(*Table Error*)
IF dwMask = 16#4A THEN
	stGroupMessage := 'Table Error: ';
	IF NC_Error_Code = 16#4A00 THEN
		stErrorMessage := 'Table ID not allowed';
	END_IF
	IF NC_Error_Code = 16#4A01 THEN
		stErrorMessage := 'Table type not allowed';
	END_IF
	IF NC_Error_Code = 16#4A02 THEN
		stErrorMessage := 'Number of lines in the table not allowed';
	END_IF
	IF NC_Error_Code = 16#4A03 THEN
		stErrorMessage := 'Number of columns in the table is not allowed';
	END_IF
	IF NC_Error_Code = 16#4A04 THEN
		stErrorMessage := 'Step size (position delta) not allowed';
	END_IF
	IF NC_Error_Code = 16#4A05 THEN
		stErrorMessage := 'Period not allowed';
	END_IF
	IF NC_Error_Code = 16#4A06 THEN
		stErrorMessage := 'Table is not monotonic';
	END_IF
	IF NC_Error_Code = 16#4A07 THEN
		stErrorMessage := 'Table sub type is not allowed';
	END_IF
	IF NC_Error_Code = 16#4A08 THEN
		stErrorMessage := 'Table interpolation type is not allowed';
	END_IF
	IF NC_Error_Code = 16#4A09 THEN
		stErrorMessage := 'Incorrect table main type';
	END_IF
	IF NC_Error_Code = 16#4A10 THEN
		stErrorMessage := 'Table initialisation';
	END_IF
	IF NC_Error_Code = 16#4A11 THEN
		stErrorMessage := 'Not enough memory';
	END_IF
	IF NC_Error_Code = 16#4A12 THEN
		stErrorMessage := 'Function not executed, function not available';
	END_IF
	IF NC_Error_Code = 16#4A13 THEN
		stErrorMessage := 'Line index not allowed';
	END_IF
	IF NC_Error_Code = 16#4A14 THEN
		stErrorMessage := 'Column index not allowed';
	END_IF
	IF NC_Error_Code = 16#4A15 THEN
		stErrorMessage := 'Number of lines not allowed';
	END_IF
	IF NC_Error_Code = 16#4A16 THEN
		stErrorMessage := 'Number of columns not allowed';
	END_IF
	IF NC_Error_Code = 16#4A17 THEN
		stErrorMessage := 'Error in scaling or in range entry';
	END_IF
	IF NC_Error_Code = 16#4A18 THEN
		stErrorMessage := 'Multi table slave out of range';
	END_IF
	IF NC_Error_Code = 16#4A19 THEN
		stErrorMessage := 'Solo table underflow';
	END_IF
	IF NC_Error_Code = 16#4A1B THEN
		stErrorMessage := 'Incorrect execution mode';
	END_IF
	IF NC_Error_Code = 16#4A1C THEN
		stErrorMessage := 'Impermissible parameter';
	END_IF
	IF NC_Error_Code = 16#4A1D THEN
		stErrorMessage := 'Fifo is empty';
	END_IF
	IF NC_Error_Code = 16#4A1E THEN
		stErrorMessage := 'Fifo is full';
	END_IF
	IF NC_Error_Code = 16#4A1F THEN
		stErrorMessage := 'Point-Index of Motion Function invalid';
	END_IF
	IF NC_Error_Code = 16#4A20 THEN
		stErrorMessage := 'No diagonalisation of  matrix';
	END_IF
	IF NC_Error_Code = 16#4A21 THEN
		stErrorMessage := 'Number of spline points to less';
	END_IF
	IF NC_Error_Code = 16#4A22 THEN
		stErrorMessage := 'Fifo must not be overwritten';
	END_IF
END_IF

(*NC-PLC Error*)
IF dwMask = 16#4B THEN
	stGroupMessage := 'NC-PLC Error: ';
	IF NC_Error_Code = 16#4B00 THEN
		stErrorMessage := 'Axis has been stopped';
	END_IF
	IF NC_Error_Code = 16#4B01 THEN
		stErrorMessage := 'Axis cannot be started';
	END_IF
	IF NC_Error_Code = 16#4B02 THEN
		stErrorMessage := 'Control mode not allowed';
	END_IF
	IF NC_Error_Code = 16#4B03 THEN
		stErrorMessage := 'Axis is not moving';
	END_IF
	IF NC_Error_Code = 16#4B04 THEN
		stErrorMessage := 'Wrong mode for RestartPosAndVelo';
	END_IF
	IF NC_Error_Code = 16#4B05 THEN
		stErrorMessage := 'Command not allowed';
	END_IF
	IF NC_Error_Code = 16#4B06 THEN
		stErrorMessage := 'Parameter not correct';
	END_IF
	IF NC_Error_Code = 16#4B07 THEN
		stErrorMessage := 'Timeout axis function block';
	END_IF
	IF NC_Error_Code = 16#4B08 THEN
		stErrorMessage := 'Axis in protected mode';
	END_IF
	IF NC_Error_Code = 16#4B09 THEN
		stErrorMessage := 'Axis is not ready';
	END_IF
	IF NC_Error_Code = 16#4B0A THEN
		stErrorMessage := 'Homing error';
	END_IF
	IF NC_Error_Code = 16#4B0B THEN
		stErrorMessage := 'Invalid definition trigger input definition';
	END_IF
	IF NC_Error_Code = 16#4B0C THEN
		stErrorMessage := 'position latch has been deactivated';
	END_IF
	IF NC_Error_Code = 16#4B0E THEN
		stErrorMessage := 'Supplement not installed';
	END_IF
	IF NC_Error_Code = 16#4B0F THEN
		stErrorMessage := 'Timeout Register Access';
	END_IF
	IF NC_Error_Code = 16#4B10 THEN
		stErrorMessage := 'M-Function request missing';
	END_IF
	IF NC_Error_Code = 16#4B11 THEN
		stErrorMessage := 'Zero shift index is out of range';
	END_IF
	IF NC_Error_Code = 16#4B12 THEN
		stErrorMessage := 'R parameter index or size is invalid';
	END_IF
	IF NC_Error_Code = 16#4B13 THEN
		stErrorMessage := 'Index for tool description is invalid';
	END_IF
	IF NC_Error_Code = 16#4B14 THEN
		stErrorMessage := 'Version of cyclic channel interface does not match to the requested function and function block, resp.';
	END_IF
	IF NC_Error_Code = 16#4B15 THEN
		stErrorMessage := 'Channel is not ready for requested function';
	END_IF
	IF NC_Error_Code = 16#4B16 THEN
		stErrorMessage := 'Requested function is not turned on';
	END_IF
	IF NC_Error_Code = 16#4B20 THEN
		stErrorMessage := 'Cannot append all axes';
	END_IF
	IF NC_Error_Code = 16#4B30 THEN
		stErrorMessage := 'Pointer invalid';
	END_IF
	IF NC_Error_Code = 16#4B31 THEN
		stErrorMessage := 'Size of  memory invalid';
	END_IF
	IF NC_Error_Code = 16#4B32 THEN
		stErrorMessage := 'Invalid cam table ID';
	END_IF
	IF NC_Error_Code = 16#4B33 THEN
		stErrorMessage := 'Invalid point ID';
	END_IF
	IF NC_Error_Code = 16#4B34 THEN
		stErrorMessage := 'Invalid number of points ';
	END_IF
	IF NC_Error_Code = 16#4B35 THEN
		stErrorMessage := 'Invalid MC table type';
	END_IF
	IF NC_Error_Code = 16#4B36 THEN
		stErrorMessage := 'Invalid number of rows';
	END_IF
	IF NC_Error_Code = 16#4B37 THEN
		stErrorMessage := 'Invalid number of columns';
	END_IF
	IF NC_Error_Code = 16#4B38 THEN
		stErrorMessage := 'Invalid Increment';
	END_IF
	IF NC_Error_Code = 16#4B40 THEN
		stErrorMessage := 'Unsupported Terminal Type';
	END_IF
	IF NC_Error_Code = 16#4B41 THEN
		stErrorMessage := 'Register Read/Write Error';
	END_IF
	IF NC_Error_Code = 16#4B42 THEN
		stErrorMessage := 'Axis is Enabled';
	END_IF
	IF NC_Error_Code = 16#4B60 THEN
		stErrorMessage := 'Motion command not be activated';
	END_IF
	IF NC_Error_Code = 16#4B61 THEN
		stErrorMessage := 'Motion command could not be monitored by the PLC';
	END_IF
	IF NC_Error_Code = 16#4B62 THEN
		stErrorMessage := 'Buffered command finished with error';
	END_IF
	IF NC_Error_Code = 16#4B63 THEN
		stErrorMessage := 'Buffered command finished without state feedback';
	END_IF
	IF NC_Error_Code = 16#4B64 THEN
		stErrorMessage := 'BufferMode not supported';
	END_IF
	IF NC_Error_Code = 16#4B71 THEN
		stErrorMessage := 'Invalid NCI Entry Type';
	END_IF
	IF NC_Error_Code = 16#4B72 THEN
		stErrorMessage := 'NciFeedTable full';
	END_IF
	IF NC_Error_Code = 16#4B74 THEN
		stErrorMessage := 'ST_NciTangentialFollowingDesc: tangential axis is not an auxiliary axis';
	END_IF
	IF NC_Error_Code = 16#4B75 THEN
		stErrorMessage := 'ST_NciTangentialFollowingDesc: nPathAxis1 and nPathAxis2, resp. are no path axes. ';
	END_IF
	IF NC_Error_Code = 16#4B76 THEN
		stErrorMessage := 'ST_NciTangentialFollwoingDesc: nPathAxis1 and nPathAxis2 are equal.';
	END_IF
	IF NC_Error_Code = 16#4B77 THEN
		stErrorMessage := 'ST_NciGeoCirclePlane';
	END_IF
	IF NC_Error_Code = 16#4B78 THEN
		stErrorMessage := 'Internal error in calculation of the tangential following';
	END_IF
	IF NC_Error_Code = 16#4B79 THEN
		stErrorMessage := 'Tangential following';
	END_IF
	IF NC_Error_Code = 16#4B7B THEN
		stErrorMessage := 'Tangential Following';
	END_IF
	IF NC_Error_Code = 16#4B7C THEN
		stErrorMessage := 'FB_NciFeedTablePreparation:  pEntry is NULL';
	END_IF
	IF NC_Error_Code = 16#4B7D THEN
		stErrorMessage := 'FB_NciFeedTablePreparation: The specified nEntryType does not match the the structure type';
	END_IF
	IF NC_Error_Code = 16#4B7E THEN
		stErrorMessage := 'ST_NciMFuncFast and ST_NciMFuncHsk';
	END_IF
	IF NC_Error_Code = 16#4B7F THEN
		stErrorMessage := 'ST_NciDynOvr';
	END_IF
	IF NC_Error_Code = 16#4B80 THEN
		stErrorMessage := 'ST_NciVertexSmoothing';
	END_IF
	IF NC_Error_Code = 16#4B81 THEN
		stErrorMessage := 'FB_NciFeedTablePrepartion';
	END_IF
END_IF

(*Finally, Concatenate Group Message and Error Message and Return*)

FUN_GTAC_NC_Error_Messages:= CONCAT(stGroupMessage, stErrorMessage);

END_FUNCTION

// ---- POUs/FUNs/FUN_GTAC_ZeroSecsInUDINT_Time.TcPOU
(*Take a var of UDINT type that is being used to store time, convert to timestruct type to check if seconds are not zero.
If not zero, round the minutes section and then zero the seconds.
Convert back to UDINT as return

original author: Brent Lekx-Toniolo of Fort Wisers

----------------------------------------------------------------------------------------------------------------------
REVISION NOTES: 
	Date: Jan, 2020:
	- initial concept, blt
------------------------------------------------------------------------------------------------------------------------
*)



FUNCTION FUN_GTAC_ZeroSecsInUDINT_Time : UDINT
VAR_INPUT

	Time_In_UDINT: UDINT;

END_VAR
VAR

	Time_In_Timestruct: Timestruct;

END_VAR

(* Convert To Timestruct *)

	Time_In_Timestruct.wHour:= UDINT_TO_WORD(Time_In_UDINT / 3600000);
	Time_In_Timestruct.wMinute:= UDINT_TO_WORD(Time_In_UDINT / 60000) - (Time_In_Timestruct.wHour*60);
	Time_In_Timestruct.wSecond:= UDINT_TO_WORD(Time_In_UDINT / 1000) - (Time_In_Timestruct.wHour*60*60) - (Time_In_Timestruct.wMinute*60);

(*Evaluate Seconds Portion*)

	IF 	Time_In_Timestruct.wSecond <>0
		THEN
		IF Time_In_Timestruct.wSecond >=30
			THEN
			(*Round minute up, then zero seconds*)
			Time_In_Timestruct.wMinute:= Time_In_Timestruct.wMinute+1;
			Time_In_Timestruct.wSecond:= 0;

		ELSIF Time_In_Timestruct.wSecond < 30
			THEN
			(*Leave Minute and simply zero seconds*)
			Time_In_Timestruct.wSecond:= 0;

		END_IF;
	END_IF;

(*Finally Return*)

	FUN_GTAC_ZeroSecsInUDINT_Time:= TOD_TO_UDINT(FUN_GTAC_TIMESTRUCTtoTOD(Time_In_Timestruct));

END_FUNCTION

// ---- POUs/Robot_InterLock_Map.TcPOU
(*!!!!!!!!!!!!!!!!!!!!!!!!!!!!!!!!!!!!!!!!!!!!!!!!!!!!!!!!!!!!!!!!!!!!!!!!!!!!!!!!!!!!!!!!!!!!!!!!!!!!!!!!!!!!!!!!!!!!!!!!!!!!!!!!!!!!!!!!!!!!!!!!!!!!!!!!!!!!
Robot Interlock Map:
	Robot to Human Interference Mapping,
	Robot to Equipment Interference Mapping,
	Robot to Robot Interference Mapping,
	Teach Interlock Mapping,
	
	auth. Brent Lekx-Toniolo of Toniolo Research & Development Inc.; 
	August 2010
----------------------------------------------------------------------------------------------------------------------
REVISION NOTES: 
	Date: October 2014
	- Added capability of up to 30 robots, b.lekx-toniolo

----------------------------------------------------------------------------------------------------------------------
General Guidlines:
 The following is just general generic concept, may not apply in each application

	HumanInterf1 - Human Tool 1 (LH side from Human)
	HumanInterf2 - Human Tool 2 (RH Side from Human)
	HumanInterf3 - Human Tool 3
	HumanInterf4 - Human Tool 4
	HumanInterf5 - Human Tool 5
	HumanInterf6 - Human Tool 6
	HumanInterf7 - Human Tool 7
	HumanInterf8 - Human Tool 8

	EquipInterf1 - Internal Tool
	EquipInterf2 - Internal Tool
	EquipInterf3 - Internal Tool
	EquipInterf4 - Internal Tool
	EquipInterf5 - Internal Ped
	EquipInterf6 - Internal Ped
	EquipInterf7 - Internal Ped
	EquipInterf8 - Reserved for: Cell Services (Master Test, Brake Test, Tip Change etc)

	RobotInterf1-8 - Robot to Robot Interf Zones

*)

PROGRAM Robot_InterLock_Map
	VAR_INPUT
		Enable_Prog: BOOL;
	END_VAR

	VAR
	(*add Internal Vars here*)
END_VAR

	VAR_OUTPUT
		Prog_Ok: BOOL;
	END_VAR

	(*Set Prog_OK to True*)
	Prog_OK:= TRUE;
(*$$$$$$$$$$$$$$$$$$$$$$$$$$$$$$$$$$$$$$$$$$$$$$$$Gather Status Of Hardware $$$$$$$$$$$$$$$$$$$$$$$$$$$$$$$$$$$$$$$$$$$$$$$$$$$$*)



(*Robot  Interference Zone Mapping, Add Robot to Robot Interference Mapping and Tool Interlocks Here*)
(*R1-----------------------------------------------------------------*)
	R1_Data.OK_ToEnter_HumanInterf1:= (Fix01.Tool_Call_ForSweepA AND Fix02.Tool_Call_ForSweepA)
									AND MAIN.R2.At_Home AND MAIN.R3.At_Home;
	R1_Data.OK_ToEnter_HumanInterf2:= (Fix01.Tool_Call_ForSweepB AND Fix02.Tool_Call_ForSweepB)
									AND MAIN.R2.At_Home AND MAIN.R3.At_Home;
	R1_Data.OK_ToEnter_HumanInterf3:= FALSE;
	R1_Data.OK_ToEnter_HumanInterf4:= FALSE;
	R1_Data.OK_ToEnter_HumanInterf5:= FALSE;
	R1_Data.OK_ToEnter_HumanInterf6:= FALSE;
	R1_Data.OK_ToEnter_HumanInterf7:= FALSE;
	R1_Data.OK_ToEnter_HumanInterf8:= FALSE;
	R1_Data.OK_ToEnter_EquipInterf1:= Fix01.Tool_Call_ForWeldRobots;
	R1_Data.OK_ToEnter_EquipInterf2:= Fix02.Tool_Call_ForWeldRobots;
	R1_Data.OK_ToEnter_EquipInterf3:= Fix01.Tool_Call_ForUnloadRobots1;
	R1_Data.OK_ToEnter_EquipInterf4:= Fix02.Tool_Call_ForUnloadRobots1;
	R1_Data.OK_ToEnter_EquipInterf5:= FALSE; 
	R1_Data.OK_ToEnter_EquipInterf6:= FALSE; 
	R1_Data.OK_ToEnter_EquipInterf7:= FALSE;
	R1_Data.OK_ToEnter_EquipInterf8:= Cell_Services_Prog.Service_Call_ForAllRobots OR Cell_Services_Prog.Service_Call_ForRobot1
							  AND NOT (Fix01.Start_TurntableA AND Fix02.Start_TurntableA)
					          AND NOT (Fix01.Start_TurntableB AND Fix02.Start_TurntableB);
	R1_Data.OK_ToEnter_EquipInterf9:= FALSE;
	R1_Data.OK_ToEnter_RobotInterfs.0:= MAIN.R2.Clear_Of_RobotInterfs.0; //105
	R1_Data.OK_ToEnter_RobotInterfs.1:= FALSE; //106
	R1_Data.OK_ToEnter_RobotInterfs.2:= FALSE; //107
	R1_Data.OK_ToEnter_RobotInterfs.3:= FALSE; //108
	R1_Data.OK_ToEnter_RobotInterfs.4:= FALSE;//R1&R2-109
	R1_Data.OK_ToEnter_RobotInterfs.5:= FALSE;//R1&R3-110
	R1_Data.OK_ToEnter_RobotInterfs.6:= MAIN.R2.Clear_Of_RobotInterfs.6;//R1&R2-111
	R1_Data.OK_ToEnter_RobotInterfs.7:= FALSE;//R1&R3-112

	(*Teach Interlocks*)
	IF GTAC_CONFIG.Under_Construction
		THEN
			R1_Data.Teach_Interlock:= TRUE;

	ELSE
			R1_Data.Teach_Interlock:= (NOT Main.R2.In_Teach AND NOT Main.R3.In_Teach) OR TRUE (*DEBUG*); (*DEBUG EXAMPLE ONLY - Add Other Robots In teach etc Interlocks here, must be held high to NOT hold this robot*)

	END_IF;

(*R2-----------------------------------------------------------------*)
	R2_Data.OK_ToEnter_HumanInterf1:= FALSE;
	R2_Data.OK_ToEnter_HumanInterf2:= FALSE;
	R2_Data.OK_ToEnter_HumanInterf3:= FALSE;
	R2_Data.OK_ToEnter_HumanInterf4:= FALSE;
	R2_Data.OK_ToEnter_HumanInterf5:= FALSE;
	R2_Data.OK_ToEnter_HumanInterf6:= FALSE;
	R2_Data.OK_ToEnter_HumanInterf7:= FALSE;
	R2_Data.OK_ToEnter_HumanInterf8:= FALSE;
	R2_Data.OK_ToEnter_EquipInterf1:= Fix01.Tool_Call_ForWeldRobots;
	R2_Data.OK_ToEnter_EquipInterf2:= Fix02.Tool_Call_ForWeldRobots;
	R2_Data.OK_ToEnter_EquipInterf3:= Fix01.Tool_Call_ForUnloadRobots1;
	R2_Data.OK_ToEnter_EquipInterf4:= Fix02.Tool_Call_ForUnloadRobots1;
	R2_Data.OK_ToEnter_EquipInterf5:= FALSE;
	R2_Data.OK_ToEnter_EquipInterf6:= FALSE;
	R2_Data.OK_ToEnter_EquipInterf7:= FALSE;
	R2_Data.OK_ToEnter_EquipInterf8:= (Cell_Services_Prog.Service_Call_ForAllRobots OR Cell_Services_Prog.Service_Call_ForRobot2)
									AND ((Fix01.TurntableA_At_Robot OR Fix01.TurntableB_At_Robot) AND Fix01.Turntable_Clear AND Fix02.Turntable_Clear)
							    AND NOT (Fix01.Start_TurntableA AND Fix02.Start_TurntableA)
								AND NOT (Fix01.Start_TurntableB AND Fix02.Start_TurntableB);
	R2_Data.OK_ToEnter_EquipInterf9:= FALSE;
	R2_Data.OK_ToEnter_RobotInterfs.0:= MAIN.R1.Clear_Of_RobotInterfs.0;
	R2_Data.OK_ToEnter_RobotInterfs.1:= MAIN.R3.Clear_Of_RobotInterfs.1;
	R2_Data.OK_ToEnter_RobotInterfs.2:= FALSE;
	R2_Data.OK_ToEnter_RobotInterfs.3:= FALSE;
	R2_Data.OK_ToEnter_RobotInterfs.4:= FALSE;
	R2_Data.OK_ToEnter_RobotInterfs.5:= FALSE;
	R2_Data.OK_ToEnter_RobotInterfs.6:= MAIN.R1.Clear_Of_RobotInterfs.6 AND MAIN.R3.Clear_Of_RobotInterfs.6;
	R2_Data.OK_ToEnter_RobotInterfs.7:= FALSE;
	
	(*Teach Interlocks*)
	IF GTAC_CONFIG.Under_Construction
		THEN
			R2_Data.Teach_Interlock:= TRUE;

	ELSE
			R2_Data.Teach_Interlock:= (NOT Main.R1.In_Teach AND NOT Main.R3.In_Teach) OR TRUE (*DEBUG*); (*DEBUG EXAMPLE ONLY - Add Other Robots In teach etc Interlocks here, must be held high to NOT hold this robot*)

	END_IF;


(*R3-----------------------------------------------------------------*)
	R3_Data.OK_ToEnter_HumanInterf1:= FALSE;
	R3_Data.OK_ToEnter_HumanInterf2:= FALSE;
	R3_Data.OK_ToEnter_HumanInterf3:= FALSE;
	R3_Data.OK_ToEnter_HumanInterf4:= FALSE;
	R3_Data.OK_ToEnter_HumanInterf5:= FALSE;
	R3_Data.OK_ToEnter_HumanInterf6:= FALSE;
	R3_Data.OK_ToEnter_HumanInterf7:= FALSE;
	R3_Data.OK_ToEnter_HumanInterf8:= FALSE;
	R3_Data.OK_ToEnter_EquipInterf1:= Fix01.Tool_Call_ForWeldRobots;
	R3_Data.OK_ToEnter_EquipInterf2:= Fix02.Tool_Call_ForWeldRobots;
	R3_Data.OK_ToEnter_EquipInterf3:= Fix01.Tool_Call_ForUnloadRobots1;
	R3_Data.OK_ToEnter_EquipInterf4:= Fix02.Tool_Call_ForUnloadRobots1;
	R3_Data.OK_ToEnter_EquipInterf5:= FALSE;
	R3_Data.OK_ToEnter_EquipInterf6:= FALSE;
	R3_Data.OK_ToEnter_EquipInterf7:= FALSE;
	R2_Data.OK_ToEnter_EquipInterf8:= (Cell_Services_Prog.Service_Call_ForAllRobots OR Cell_Services_Prog.Service_Call_ForRobot2)
									AND ((Fix01.TurntableA_At_Robot OR Fix01.TurntableB_At_Robot) AND Fix01.Turntable_Clear AND Fix02.Turntable_Clear)
							    AND NOT (Fix01.Start_TurntableA AND Fix02.Start_TurntableA)
								AND NOT (Fix01.Start_TurntableB AND Fix02.Start_TurntableB);
	R3_Data.OK_ToEnter_EquipInterf9:= FALSE;
	R3_Data.OK_ToEnter_RobotInterfs.0:= FALSE;
	R3_Data.OK_ToEnter_RobotInterfs.1:= MAIN.R2.Clear_Of_RobotInterfs.1;
	R3_Data.OK_ToEnter_RobotInterfs.2:= FALSE;
	R3_Data.OK_ToEnter_RobotInterfs.3:= FALSE;
	R3_Data.OK_ToEnter_RobotInterfs.4:= FALSE;
	R3_Data.OK_ToEnter_RobotInterfs.5:= FALSE;
	R3_Data.OK_ToEnter_RobotInterfs.6:= MAIN.R2.Clear_Of_RobotInterfs.6;
	R3_Data.OK_ToEnter_RobotInterfs.7:= FALSE;

	(*Teach Interlocks*)
	IF GTAC_CONFIG.Under_Construction
		THEN
			R3_Data.Teach_Interlock:= TRUE;

	ELSE
			R3_Data.Teach_Interlock:= (NOT Main.R1.In_Teach AND NOT Main.R2.In_Teach) OR TRUE (*DEBUG*); (*DEBUG EXAMPLE ONLY - Add Other Robots In teach etc Interlocks here, must be held high to NOT hold this robot*)

	END_IF;


(*R4-----------------------------------------------------------------*)
	R4_Data.OK_ToEnter_HumanInterf1:= Fix05.Tool_Call_ForLoadRobots1;
	R4_Data.OK_ToEnter_HumanInterf2:= FALSE;
	R4_Data.OK_ToEnter_HumanInterf3:= FALSE;
	R4_Data.OK_ToEnter_HumanInterf4:= FALSE;
	R4_Data.OK_ToEnter_HumanInterf5:= FALSE;
	R4_Data.OK_ToEnter_HumanInterf6:= FALSE;
	R4_Data.OK_ToEnter_HumanInterf7:= FALSE;
	R4_Data.OK_ToEnter_HumanInterf8:= FALSE;
	R4_Data.OK_ToEnter_EquipInterf1:= (Fix01.Tool_Call_ForUnloadRobots1 OR  Fix02.Tool_Call_ForUnloadRobots1) AND Fix101.All_Sensors_Off; //9 (*Dont pick up off Fix01 or 02 unless Fix101 is ready to receive*)
	R4_Data.OK_ToEnter_EquipInterf2:= Fix101.Tool_Call_ForLoadRobots1 OR Fix101.Tool_Call_ForUnloadRobots1; //10
	R4_Data.OK_ToEnter_EquipInterf3:= Fix03.Tool_Call_ForLoadRobots1 OR Fix04.Tool_Call_ForLoadRobots1 OR (Fix102.All_Sensors_Off AND (Fix03.Tool_Call_ForUnloadRobots1 OR Fix04.Tool_Call_ForUnloadRobots1)); //11 (*Dont pick up off Fix03 or 04 unless Fix102 is ready to receive*) //11 
	R4_Data.OK_ToEnter_EquipInterf4:= Fix102.Tool_Call_ForLoadRobots1 OR Fix102.Tool_Call_ForUnloadRobots1;//12
	R4_Data.OK_ToEnter_EquipInterf5:= Fix103.Tool_Call_ForLoadRobots1; //13
	R4_Data.OK_ToEnter_EquipInterf6:= Fix104.Tool_Call_ForLoadRobots1; //14
	R4_Data.OK_ToEnter_EquipInterf7:= Fix105.Tool_Call_ForLoadRobots1; //15
	R4_Data.OK_ToEnter_EquipInterf8:= Cell_Services_Prog.Service_Call_ForAllRobots OR Cell_Services_Prog.Service_Call_ForRobot4; //16
	R4_Data.OK_ToEnter_EquipInterf9:= MAIN.PED[1].Tool_Call_ForWorkRobots;//17
	R4_Data.OK_ToEnter_RobotInterfs.0:= FALSE;
	R4_Data.OK_ToEnter_RobotInterfs.1:= FALSE;
	R4_Data.OK_ToEnter_RobotInterfs.2:= FALSE;
	R4_Data.OK_ToEnter_RobotInterfs.3:= FALSE;
	R4_Data.OK_ToEnter_RobotInterfs.4:= FALSE;
	R4_Data.OK_ToEnter_RobotInterfs.5:= FALSE;
	R4_Data.OK_ToEnter_RobotInterfs.6:= FALSE;
	R4_Data.OK_ToEnter_RobotInterfs.7:= FALSE;

	(*Teach Interlocks*)
	IF GTAC_CONFIG.Under_Construction
		THEN
			R4_Data.Teach_Interlock:= TRUE;

	ELSE
			R4_Data.Teach_Interlock:= TRUE; (*DEBUG - Add Other Robots In teach etc Interlocks here, must be held high to NOT hold this robot*)

	END_IF;


(*R5-----------------------------------------------------------------*)
	R5_Data.OK_ToEnter_HumanInterf1:= (Fix03.Tool_Call_ForSweepA AND Fix04.Tool_Call_ForSweepA)
									AND MAIN.R6.At_Home;
	R5_Data.OK_ToEnter_HumanInterf2:= (Fix03.Tool_Call_ForSweepB AND Fix04.Tool_Call_ForSweepB)
									AND MAIN.R6.At_Home;
	R5_Data.OK_ToEnter_HumanInterf3:= FALSE;
	R5_Data.OK_ToEnter_HumanInterf4:= FALSE;
	R5_Data.OK_ToEnter_HumanInterf5:= FALSE;
	R5_Data.OK_ToEnter_HumanInterf6:= FALSE;
	R5_Data.OK_ToEnter_HumanInterf7:= FALSE;
	R5_Data.OK_ToEnter_HumanInterf8:= FALSE;
	R5_Data.OK_ToEnter_EquipInterf1:= Fix03.Tool_Call_ForWeldRobots;
	R5_Data.OK_ToEnter_EquipInterf2:= Fix04.Tool_Call_ForWeldRobots;
	R5_Data.OK_ToEnter_EquipInterf3:= Fix03.Tool_Call_ForLoadRobots1;
	R5_Data.OK_ToEnter_EquipInterf4:= Fix04.Tool_Call_ForLoadRobots1;
	R5_Data.OK_ToEnter_EquipInterf5:= FALSE;
	R5_Data.OK_ToEnter_EquipInterf6:= FALSE;
	R5_Data.OK_ToEnter_EquipInterf7:= FALSE;
	R5_Data.OK_ToEnter_EquipInterf8:= Cell_Services_Prog.Service_Call_ForAllRobots OR Cell_Services_Prog.Service_Call_ForRobot5;
	R5_Data.OK_ToEnter_EquipInterf9:= FALSE;
	R5_Data.OK_ToEnter_RobotInterfs.0:= MAIN.R6.Clear_Of_RobotInterfs.0; //105
	R5_Data.OK_ToEnter_RobotInterfs.1:= MAIN.R6.Clear_Of_RobotInterfs.1; //106
	R5_Data.OK_ToEnter_RobotInterfs.2:= MAIN.R6.Clear_Of_RobotInterfs.2; //107
	R5_Data.OK_ToEnter_RobotInterfs.3:= MAIN.R6.Clear_Of_RobotInterfs.3; //108
	R5_Data.OK_ToEnter_RobotInterfs.4:= MAIN.R6.Clear_Of_RobotInterfs.4; //109
	R5_Data.OK_ToEnter_RobotInterfs.5:= MAIN.R6.Clear_Of_RobotInterfs.5; //110
	R5_Data.OK_ToEnter_RobotInterfs.6:= MAIN.R6.Clear_Of_RobotInterfs.6; //111
	R5_Data.OK_ToEnter_RobotInterfs.7:= MAIN.R6.Clear_Of_RobotInterfs.7; //112

	(*Teach Interlocks*)
	IF GTAC_CONFIG.Under_Construction
		THEN
			R5_Data.Teach_Interlock:= TRUE;

	ELSE
			R5_Data.Teach_Interlock:= TRUE; (*DEBUG - Add Other Robots In teach etc Interlocks here, must be held high to NOT hold this robot*)

	END_IF;


(*R6-----------------------------------------------------------------*)
	R6_Data.OK_ToEnter_HumanInterf1:= FALSE;
	R6_Data.OK_ToEnter_HumanInterf2:= FALSE;
	R6_Data.OK_ToEnter_HumanInterf3:= FALSE;
	R6_Data.OK_ToEnter_HumanInterf4:= FALSE;
	R6_Data.OK_ToEnter_HumanInterf5:= FALSE;
	R6_Data.OK_ToEnter_HumanInterf6:= FALSE;
	R6_Data.OK_ToEnter_HumanInterf7:= FALSE;
	R6_Data.OK_ToEnter_HumanInterf8:= FALSE;
	R6_Data.OK_ToEnter_EquipInterf1:= Fix03.Tool_Call_ForWeldRobots;
	R6_Data.OK_ToEnter_EquipInterf2:= Fix04.Tool_Call_ForWeldRobots;
	R6_Data.OK_ToEnter_EquipInterf3:= Fix03.Tool_Call_ForLoadRobots1;
	R6_Data.OK_ToEnter_EquipInterf4:= Fix04.Tool_Call_ForLoadRobots1;
	R6_Data.OK_ToEnter_EquipInterf5:= FALSE;
	R6_Data.OK_ToEnter_EquipInterf6:= FALSE;
	R6_Data.OK_ToEnter_EquipInterf7:= FALSE;
	R6_Data.OK_ToEnter_EquipInterf8:=  Cell_Services_Prog.Service_Call_ForAllRobots OR Cell_Services_Prog.Service_Call_ForRobot6;
	R6_Data.OK_ToEnter_EquipInterf9:= FALSE;
	R6_Data.OK_ToEnter_RobotInterfs.0:= MAIN.R5.Clear_Of_RobotInterfs.0; //105
	R6_Data.OK_ToEnter_RobotInterfs.1:= MAIN.R5.Clear_Of_RobotInterfs.1; //106
	R6_Data.OK_ToEnter_RobotInterfs.2:= MAIN.R5.Clear_Of_RobotInterfs.2; //107
	R6_Data.OK_ToEnter_RobotInterfs.3:= MAIN.R5.Clear_Of_RobotInterfs.3; //108
	R6_Data.OK_ToEnter_RobotInterfs.4:= MAIN.R5.Clear_Of_RobotInterfs.4; //109
	R6_Data.OK_ToEnter_RobotInterfs.5:= MAIN.R5.Clear_Of_RobotInterfs.5; //110
	R6_Data.OK_ToEnter_RobotInterfs.6:= MAIN.R5.Clear_Of_RobotInterfs.6; //111
	R6_Data.OK_ToEnter_RobotInterfs.7:= MAIN.R5.Clear_Of_RobotInterfs.7; //112

	(*Teach Interlocks*)
	IF GTAC_CONFIG.Under_Construction
		THEN
			R6_Data.Teach_Interlock:= TRUE;

	ELSE
			R6_Data.Teach_Interlock:= TRUE; (*DEBUG - Add Other Robots In teach etc Interlocks here, must be held high to NOT hold this robot*)

	END_IF;


(*R7-----------------------------------------------------------------*)
	R7_Data.OK_ToEnter_HumanInterf1:= FALSE;
	R7_Data.OK_ToEnter_HumanInterf2:= FALSE;
	R7_Data.OK_ToEnter_HumanInterf3:= FALSE;
	R7_Data.OK_ToEnter_HumanInterf4:= FALSE;
	R7_Data.OK_ToEnter_HumanInterf5:= FALSE;
	R7_Data.OK_ToEnter_HumanInterf6:= FALSE;
	R7_Data.OK_ToEnter_HumanInterf7:= FALSE;
	R7_Data.OK_ToEnter_HumanInterf8:= FALSE;
	R7_Data.OK_ToEnter_EquipInterf1:= Fix101.Tool_Call_ForWeldRobots;
	R7_Data.OK_ToEnter_EquipInterf2:= Fix101.Tool_Call_ForSweepA;
	R7_Data.OK_ToEnter_EquipInterf3:= FALSE;
	R7_Data.OK_ToEnter_EquipInterf4:= FALSE;
	R7_Data.OK_ToEnter_EquipInterf5:= FALSE;
	R7_Data.OK_ToEnter_EquipInterf6:= FALSE;
	R7_Data.OK_ToEnter_EquipInterf7:= FALSE;
	R7_Data.OK_ToEnter_EquipInterf8:=  Cell_Services_Prog.Service_Call_ForAllRobots OR Cell_Services_Prog.Service_Call_ForRobot7;
	R7_Data.OK_ToEnter_EquipInterf9:= FALSE;
	R7_Data.OK_ToEnter_RobotInterfs.0:= MAIN.R8.Clear_Of_RobotInterfs.0 AND MAIN.R9.Clear_Of_RobotInterfs.0;//105
	R7_Data.OK_ToEnter_RobotInterfs.1:= MAIN.R8.Clear_Of_RobotInterfs.1 AND MAIN.R9.Clear_Of_RobotInterfs.1;//106
	R7_Data.OK_ToEnter_RobotInterfs.2:= MAIN.R8.Clear_Of_RobotInterfs.2 AND MAIN.R9.Clear_Of_RobotInterfs.2;//107
	R7_Data.OK_ToEnter_RobotInterfs.3:= MAIN.R8.Clear_Of_RobotInterfs.3 AND MAIN.R9.Clear_Of_RobotInterfs.3;//108
	R7_Data.OK_ToEnter_RobotInterfs.4:= MAIN.R8.Clear_Of_RobotInterfs.4;//109
	R7_Data.OK_ToEnter_RobotInterfs.5:= MAIN.R8.Clear_Of_RobotInterfs.5;//110
	R7_Data.OK_ToEnter_RobotInterfs.6:= MAIN.R8.Clear_Of_RobotInterfs.6;//111
	R7_Data.OK_ToEnter_RobotInterfs.7:= MAIN.R9.Clear_Of_RobotInterfs.7;//112

	(*Teach Interlocks*)
	IF GTAC_CONFIG.Under_Construction
		THEN
			R7_Data.Teach_Interlock:= TRUE;

	ELSE
			R7_Data.Teach_Interlock:= TRUE; (*DEBUG - Add Other Robots In teach etc Interlocks here, must be held high to NOT hold this robot*)

	END_IF;


(*R8-----------------------------------------------------------------*)
	R8_Data.OK_ToEnter_HumanInterf1:= FALSE;
	R8_Data.OK_ToEnter_HumanInterf2:= FALSE;
	R8_Data.OK_ToEnter_HumanInterf3:= FALSE;
	R8_Data.OK_ToEnter_HumanInterf4:= FALSE;
	R8_Data.OK_ToEnter_HumanInterf5:= FALSE;
	R8_Data.OK_ToEnter_HumanInterf6:= FALSE;
	R8_Data.OK_ToEnter_HumanInterf7:= FALSE;
	R8_Data.OK_ToEnter_HumanInterf8:= FALSE;
	R8_Data.OK_ToEnter_EquipInterf1:= Fix101.Tool_Call_ForWeldRobots;
	R8_Data.OK_ToEnter_EquipInterf2:= FALSE;
	R8_Data.OK_ToEnter_EquipInterf3:= FALSE;
	R8_Data.OK_ToEnter_EquipInterf4:= FALSE;
	R8_Data.OK_ToEnter_EquipInterf5:= FALSE;
	R8_Data.OK_ToEnter_EquipInterf6:= FALSE;
	R8_Data.OK_ToEnter_EquipInterf7:= FALSE;
	R8_Data.OK_ToEnter_EquipInterf8:=  Cell_Services_Prog.Service_Call_ForAllRobots OR Cell_Services_Prog.Service_Call_ForRobot8;
	R8_Data.OK_ToEnter_EquipInterf9:= FALSE;
	R8_Data.OK_ToEnter_RobotInterfs.0:= MAIN.R7.Clear_Of_RobotInterfs.0;//105
	R8_Data.OK_ToEnter_RobotInterfs.1:= MAIN.R7.Clear_Of_RobotInterfs.1;//106
	R8_Data.OK_ToEnter_RobotInterfs.2:= MAIN.R7.Clear_Of_RobotInterfs.2;//107
	R8_Data.OK_ToEnter_RobotInterfs.3:= MAIN.R7.Clear_Of_RobotInterfs.4;//R8-108 <-> R7 -109
	R8_Data.OK_ToEnter_RobotInterfs.4:= MAIN.R7.Clear_Of_RobotInterfs.5;//R8-109 <-> R7 -110
	R8_Data.OK_ToEnter_RobotInterfs.5:= MAIN.R7.Clear_Of_RobotInterfs.6;//R8-110 <-> R7 -111
	R8_Data.OK_ToEnter_RobotInterfs.6:= MAIN.R9.Clear_Of_RobotInterfs.4;//R8-111 <-> R9 -109
	R8_Data.OK_ToEnter_RobotInterfs.7:= MAIN.R9.Clear_Of_RobotInterfs.5;//R8-112 <-> R9 -110

	(*Teach Interlocks*)
	IF GTAC_CONFIG.Under_Construction
		THEN
			R8_Data.Teach_Interlock:= TRUE;

	ELSE
			R8_Data.Teach_Interlock:= TRUE; (*DEBUG - Add Other Robots In teach etc Interlocks here, must be held high to NOT hold this robot*)

	END_IF;


(*R9-----------------------------------------------------------------*)
	R9_Data.OK_ToEnter_HumanInterf1:= FALSE;
	R9_Data.OK_ToEnter_HumanInterf2:= FALSE;
	R9_Data.OK_ToEnter_HumanInterf3:= FALSE;
	R9_Data.OK_ToEnter_HumanInterf4:= FALSE;
	R9_Data.OK_ToEnter_HumanInterf5:= FALSE;
	R9_Data.OK_ToEnter_HumanInterf6:= FALSE;
	R9_Data.OK_ToEnter_HumanInterf7:= FALSE;
	R9_Data.OK_ToEnter_HumanInterf8:= FALSE;
	R9_Data.OK_ToEnter_EquipInterf1:= Fix101.Tool_Call_ForWeldRobots;
	R9_Data.OK_ToEnter_EquipInterf2:= FALSE;
	R9_Data.OK_ToEnter_EquipInterf3:= FALSE;
	R9_Data.OK_ToEnter_EquipInterf4:= FALSE;
	R9_Data.OK_ToEnter_EquipInterf5:= FALSE;
	R9_Data.OK_ToEnter_EquipInterf6:= FALSE;
	R9_Data.OK_ToEnter_EquipInterf7:= FALSE;
	R9_Data.OK_ToEnter_EquipInterf8:=  Cell_Services_Prog.Service_Call_ForAllRobots OR Cell_Services_Prog.Service_Call_ForRobot9;
	R9_Data.OK_ToEnter_EquipInterf9:= FALSE;
	R9_Data.OK_ToEnter_RobotInterfs.0:= MAIN.R7.Clear_Of_RobotInterfs.0;//105
	R9_Data.OK_ToEnter_RobotInterfs.1:= MAIN.R7.Clear_Of_RobotInterfs.1;//106
	R9_Data.OK_ToEnter_RobotInterfs.2:= MAIN.R7.Clear_Of_RobotInterfs.2;//107
	R9_Data.OK_ToEnter_RobotInterfs.3:= MAIN.R8.Clear_Of_RobotInterfs.3;//108
	R9_Data.OK_ToEnter_RobotInterfs.4:= MAIN.R8.Clear_Of_RobotInterfs.4;//109
	R9_Data.OK_ToEnter_RobotInterfs.5:= MAIN.R8.Clear_Of_RobotInterfs.5;//110
	R9_Data.OK_ToEnter_RobotInterfs.6:= FALSE;
	R9_Data.OK_ToEnter_RobotInterfs.7:= MAIN.R7.Clear_Of_RobotInterfs.7;//112

	(*Teach Interlocks*)
	IF GTAC_CONFIG.Under_Construction
		THEN
			R9_Data.Teach_Interlock:= TRUE;

	ELSE
			R9_Data.Teach_Interlock:= TRUE; (*DEBUG - Add Other Robots In teach etc Interlocks here, must be held high to NOT hold this robot*)

	END_IF;


(*R10-----------------------------------------------------------------*)
	R10_Data.OK_ToEnter_HumanInterf1:= FALSE;
	R10_Data.OK_ToEnter_HumanInterf2:= FALSE;
	R10_Data.OK_ToEnter_HumanInterf3:= FALSE;
	R10_Data.OK_ToEnter_HumanInterf4:= FALSE;
	R10_Data.OK_ToEnter_HumanInterf5:= FALSE;
	R10_Data.OK_ToEnter_HumanInterf6:= FALSE;
	R10_Data.OK_ToEnter_HumanInterf7:= FALSE;
	R10_Data.OK_ToEnter_HumanInterf8:= FALSE;
	R10_Data.OK_ToEnter_EquipInterf1:= Fix102.Tool_Call_ForWeldRobots;
	R10_Data.OK_ToEnter_EquipInterf2:= Fix102.Tool_Call_ForSweepA;
	R10_Data.OK_ToEnter_EquipInterf3:= FALSE;
	R10_Data.OK_ToEnter_EquipInterf4:= FALSE;
	R10_Data.OK_ToEnter_EquipInterf5:= FALSE;
	R10_Data.OK_ToEnter_EquipInterf6:= FALSE;
	R10_Data.OK_ToEnter_EquipInterf7:= FALSE;
	R10_Data.OK_ToEnter_EquipInterf8:=  Cell_Services_Prog.Service_Call_ForAllRobots OR Cell_Services_Prog.Service_Call_ForRobot10;
	R10_Data.OK_ToEnter_EquipInterf9:= FALSE;
	R10_Data.OK_ToEnter_RobotInterfs.0:= MAIN.R11.Clear_Of_RobotInterfs.0; //105
	R10_Data.OK_ToEnter_RobotInterfs.1:= MAIN.R11.Clear_Of_RobotInterfs.1; //106
	R10_Data.OK_ToEnter_RobotInterfs.2:= MAIN.R11.Clear_Of_RobotInterfs.2; //107
	R10_Data.OK_ToEnter_RobotInterfs.3:= FALSE;
	R10_Data.OK_ToEnter_RobotInterfs.4:= FALSE;
	R10_Data.OK_ToEnter_RobotInterfs.5:= FALSE;
	R10_Data.OK_ToEnter_RobotInterfs.6:= FALSE;
	R10_Data.OK_ToEnter_RobotInterfs.7:= FALSE;

	(*Teach Interlocks*)
	IF GTAC_CONFIG.Under_Construction
		THEN
			R10_Data.Teach_Interlock:= TRUE;

	ELSE
			R10_Data.Teach_Interlock:= TRUE; (*DEBUG - Add Other Robots In teach etc Interlocks here, must be held high to NOT hold this robot*)

	END_IF;


(*R11-----------------------------------------------------------------*)
	R11_Data.OK_ToEnter_HumanInterf1:= FALSE;
	R11_Data.OK_ToEnter_HumanInterf2:= FALSE;
	R11_Data.OK_ToEnter_HumanInterf3:= FALSE;
	R11_Data.OK_ToEnter_HumanInterf4:= FALSE;
	R11_Data.OK_ToEnter_HumanInterf5:= FALSE;
	R11_Data.OK_ToEnter_HumanInterf6:= FALSE;
	R11_Data.OK_ToEnter_HumanInterf7:= FALSE;
	R11_Data.OK_ToEnter_HumanInterf8:= FALSE;
	R11_Data.OK_ToEnter_EquipInterf1:= Fix102.Tool_Call_ForWeldRobots;
	R11_Data.OK_ToEnter_EquipInterf2:= FALSE;
	R11_Data.OK_ToEnter_EquipInterf3:= FALSE;
	R11_Data.OK_ToEnter_EquipInterf4:= FALSE;
	R11_Data.OK_ToEnter_EquipInterf5:= FALSE;
	R11_Data.OK_ToEnter_EquipInterf6:= FALSE;
	R11_Data.OK_ToEnter_EquipInterf7:= FALSE;
	R11_Data.OK_ToEnter_EquipInterf8:=  Cell_Services_Prog.Service_Call_ForAllRobots OR Cell_Services_Prog.Service_Call_ForRobot11;
	R11_Data.OK_ToEnter_EquipInterf9:= FALSE;
	R11_Data.OK_ToEnter_RobotInterfs.0:= MAIN.R10.Clear_Of_RobotInterfs.0; //105
	R11_Data.OK_ToEnter_RobotInterfs.1:= MAIN.R10.Clear_Of_RobotInterfs.1; //106
	R11_Data.OK_ToEnter_RobotInterfs.2:= MAIN.R10.Clear_Of_RobotInterfs.2; //107
	R11_Data.OK_ToEnter_RobotInterfs.3:= FALSE;
	R11_Data.OK_ToEnter_RobotInterfs.4:= FALSE;
	R11_Data.OK_ToEnter_RobotInterfs.5:= FALSE;
	R11_Data.OK_ToEnter_RobotInterfs.6:= FALSE;
	R11_Data.OK_ToEnter_RobotInterfs.7:= FALSE;

	(*Teach Interlocks*)
	IF GTAC_CONFIG.Under_Construction
		THEN
			R11_Data.Teach_Interlock:= TRUE;

	ELSE
			R11_Data.Teach_Interlock:= TRUE; (*DEBUG - Add Other Robots In teach etc Interlocks here, must be held high to NOT hold this robot*)

	END_IF;

END_PROGRAM

// ---- POUs/Misc/Cell_Services_Prog.TcPOU
(*!!!!!!!!!!!!!!!!!!!!!!!!!!!!!!!!!!!!!!!!!!!!!!!!!!!!!!!!!!!!!!!!!!!!!!!!!!!!!!!!!!!!!!!!!!!!!!!!!!!!!!!!!!!!!!!!!!!!!!!!!!!!!!!!!!!!!!!!!!!!!!!!!!!!!!!!!!
Program Used to handle all Ancillary Service Requests for All Robots
Service Requests include Mastering Test, Brake Test, Tip Change and Tip Dress
	author: Brent Lekx-Toniolo of Sodecia GTAC
	July, 2013
--------------------------------------------------------------------------------------------------------------
REVISION NOTES:
	Date: October 2014
	- Added capability of up to 30 robots, b.lekx-toniolo
	Date: December 2014
 	- changed All_Robots_Clear MAIN.Rx.Task_ID_Ack from 250 to 350, b.lekx-toniolo
 	- added NOT  GTAC_CONFIG.Under_Construction TO Robot_Reqs_masterTest and BrakeTest and TipChange, JVD
	Date: March 2015
	- added/changed code to force Master and Brake Test Ext and allow all robots to ack such before starting full master or brake tests, blt
	Date: May 2016
	- added config data to auto configure code, b.lekx-toniolo (blt)
	Date: June 2017
	- broke out IF formatiing in task_id code, b.lekx-toniolo (blt)
	Date:May 2021 
	-Cleaned up Steppers Reset  to ensure that ALL steppers that are enabled are checked (CD)
	-Cleaned up Tip Change Requests to be easier to read and troubleshoot (CD)
	Date: June 2024
	- Massaged in TraccTCP code developed / tested by Wes Griffiths on project 2302901 (blt)
	Date: Sept 2024
	- Correction to Start brake Test code as per SSCC610 GH Issues #140, (blt and wg)
--------------------------------------------------------------------------------------------------------------
*)

PROGRAM Cell_Services_Prog
	VAR_INPUT
		Enable_Prog: BOOL;
		Enable_Motion: BOOL;
		Discrete_In: udt_FixXX_Input_Image_20180202;
		Dry_Cycle: BOOL;
		Cell_In_Services: BOOL;
	END_VAR

	VAR
(*Hardware Related Data Types*)


(*Standard Internal Variables*)

		(*General Internals*)
		In_Auto: BOOL;
		In_Manual: BOOL;

		Auto_Run: BOOL;
		Reset_All_Completes:BOOL;
		All_Robots_Clear: BOOL;
		All_Robots_WorkingOK: BOOL;
		All_Robots_Complete: BOOL;
		All_Robots_SteppersRST: BOOL;
		Start_All_MTRobots: BOOL;
		All_MTRobots_Proceed: BOOL;
		Start_All_BTRobots: BOOL;
		All_BTRobots_Proceed: BOOL;
		Start_All_TCRobots: BOOL;
		All_TCRobots_Proceed: BOOL;
		Start_All_TDRobots: BOOL;
		All_TDRobots_Proceed: BOOL;
		
		(*Custom for CCB*)
		Start_All_TraccTCP: BOOL;
		All_TraccTCP_Proceed: BOOL;
		
		Start_TDRobot_1: BOOL;
		Start_TDRobot_2: BOOL;
		Start_TDRobot_3: BOOL;
		Start_TDRobot_4: BOOL;
		Start_TDRobot_5: BOOL;
		Start_TDRobot_6: BOOL;
		Start_TDRobot_7: BOOL;
		Start_TDRobot_8: BOOL;
		Start_TDRobot_9: BOOL;
		Start_TDRobot_10: BOOL;
		Start_TDRobot_11: BOOL;
		Start_TDRobot_12: BOOL;
		Start_TDRobot_13: BOOL;
		Start_TDRobot_14: BOOL;
		Start_TDRobot_15: BOOL;
		Start_TDRobot_16: BOOL;
		Start_TDRobot_17: BOOL;
		Start_TDRobot_18: BOOL;
		Start_TDRobot_19: BOOL;
		Start_TDRobot_20: BOOL;
		Start_TDRobot_21: BOOL;
		Start_TDRobot_22: BOOL;
		Start_TDRobot_23: BOOL;
		Start_TDRobot_24: BOOL;
		Start_TDRobot_25: BOOL;
		Start_TDRobot_26: BOOL;
		Start_TDRobot_27: BOOL;
		Start_TDRobot_28: BOOL;
		Start_TDRobot_29: BOOL;
		Start_TDRobot_30: BOOL;

		TDRobot_1_Proceed: BOOL;
		TDRobot_2_Proceed: BOOL;
		TDRobot_3_Proceed: BOOL;
		TDRobot_4_Proceed: BOOL;
		TDRobot_5_Proceed: BOOL;
		TDRobot_6_Proceed: BOOL;
		TDRobot_7_Proceed: BOOL;
		TDRobot_8_Proceed: BOOL;
		TDRobot_9_Proceed: BOOL;
		TDRobot_10_Proceed: BOOL;
		TDRobot_11_Proceed: BOOL;
		TDRobot_12_Proceed: BOOL;
		TDRobot_13_Proceed: BOOL;
		TDRobot_14_Proceed: BOOL;
		TDRobot_15_Proceed: BOOL;
		TDRobot_16_Proceed: BOOL;
		TDRobot_17_Proceed: BOOL;
		TDRobot_18_Proceed: BOOL;
		TDRobot_19_Proceed: BOOL;
		TDRobot_20_Proceed: BOOL;
		TDRobot_21_Proceed: BOOL;
		TDRobot_22_Proceed: BOOL;
		TDRobot_23_Proceed: BOOL;
		TDRobot_24_Proceed: BOOL;
		TDRobot_25_Proceed: BOOL;
		TDRobot_26_Proceed: BOOL;
		TDRobot_27_Proceed: BOOL;
		TDRobot_28_Proceed: BOOL;
		TDRobot_29_Proceed: BOOL;
		TDRobot_30_Proceed: BOOL;
		
		(*Custom to CCB*)
		Start_TraccTCP_1: BOOL;
		Start_TraccTCP_2: BOOL;
		Start_TraccTCP_3: BOOL;
		Start_TraccTCP_4: BOOL;
		Start_TraccTCP_5: BOOL;
		Start_TraccTCP_6: BOOL;
		Start_TraccTCP_7: BOOL;
		Start_TraccTCP_8: BOOL;
		Start_TraccTCP_9: BOOL;
		Start_TraccTCP_10: BOOL;
		Start_TraccTCP_11: BOOL;
		Start_TraccTCP_12: BOOL;
		Start_TraccTCP_13: BOOL;
		Start_TraccTCP_14: BOOL;
		Start_TraccTCP_15: BOOL;
		Start_TraccTCP_16: BOOL;
		Start_TraccTCP_17: BOOL;
		Start_TraccTCP_18: BOOL;
		Start_TraccTCP_19: BOOL;
		Start_TraccTCP_20: BOOL;
		Start_TraccTCP_21: BOOL;
		Start_TraccTCP_22: BOOL;
		Start_TraccTCP_23: BOOL;
		Start_TraccTCP_24: BOOL;
		Start_TraccTCP_25: BOOL;
		Start_TraccTCP_26: BOOL;
		Start_TraccTCP_27: BOOL;
		Start_TraccTCP_28: BOOL;
		Start_TraccTCP_29: BOOL;
		Start_TraccTCP_30: BOOL;
		TraccRobot_1_Proceed: BOOL;
		TraccRobot_2_Proceed: BOOL;
		TraccRobot_3_Proceed: BOOL;
		TraccRobot_4_Proceed: BOOL;
		TraccRobot_5_Proceed: BOOL;
		TraccRobot_6_Proceed: BOOL;
		TraccRobot_7_Proceed: BOOL;
		TraccRobot_8_Proceed: BOOL;
		TraccRobot_9_Proceed: BOOL;
		TraccRobot_10_Proceed: BOOL;
		TraccRobot_11_Proceed: BOOL;
		TraccRobot_12_Proceed: BOOL;
		TraccRobot_13_Proceed: BOOL;
		TraccRobot_14_Proceed: BOOL;
		TraccRobot_15_Proceed: BOOL;
		TraccRobot_16_Proceed: BOOL;
		TraccRobot_17_Proceed: BOOL;
		TraccRobot_18_Proceed: BOOL;
		TraccRobot_19_Proceed: BOOL;
		TraccRobot_20_Proceed: BOOL;
		TraccRobot_21_Proceed: BOOL;
		TraccRobot_22_Proceed: BOOL;
		TraccRobot_23_Proceed: BOOL;
		TraccRobot_24_Proceed: BOOL;
		TraccRobot_25_Proceed: BOOL;
		TraccRobot_26_Proceed: BOOL;
		TraccRobot_27_Proceed: BOOL;
		TraccRobot_28_Proceed: BOOL;
		TraccRobot_29_Proceed: BOOL;
		TraccRobot_30_Proceed: BOOL;
		

		Robot_Reqs_TipDress: BOOL;
		Robot1_Reqs_TipDress: BOOL;
		Robot2_Reqs_TipDress: BOOL;
		Robot3_Reqs_TipDress: BOOL;
		Robot4_Reqs_TipDress: BOOL;
		Robot5_Reqs_TipDress: BOOL;
		Robot6_Reqs_TipDress: BOOL;
		Robot7_Reqs_TipDress: BOOL;
		Robot8_Reqs_TipDress: BOOL;
		Robot9_Reqs_TipDress: BOOL;
		Robot10_Reqs_TipDress: BOOL;
		Robot11_Reqs_TipDress: BOOL;
		Robot12_Reqs_TipDress: BOOL;
		Robot13_Reqs_TipDress: BOOL;
		Robot14_Reqs_TipDress: BOOL;
		Robot15_Reqs_TipDress: BOOL;
		Robot16_Reqs_TipDress: BOOL;
		Robot17_Reqs_TipDress: BOOL;
		Robot18_Reqs_TipDress: BOOL;
		Robot19_Reqs_TipDress: BOOL;
		Robot20_Reqs_TipDress: BOOL;
		Robot21_Reqs_TipDress: BOOL;
		Robot22_Reqs_TipDress: BOOL;
		Robot23_Reqs_TipDress: BOOL;
		Robot24_Reqs_TipDress: BOOL;
		Robot25_Reqs_TipDress: BOOL;
		Robot26_Reqs_TipDress: BOOL;
		Robot27_Reqs_TipDress: BOOL;
		Robot28_Reqs_TipDress: BOOL;
		Robot29_Reqs_TipDress: BOOL;
		Robot30_Reqs_TipDress: BOOL;
		
		(*Custom for CCB*)
		Robot_Reqs_TraccTCP: BOOL;
		Robot1_Reqs_TraccTCP: BOOL;
		Robot2_Reqs_TraccTCP: BOOL;
		Robot3_Reqs_TraccTCP: BOOL;
		Robot4_Reqs_TraccTCP: BOOL;
		Robot5_Reqs_TraccTCP: BOOL;
		Robot6_Reqs_TraccTCP: BOOL;
		Robot7_Reqs_TraccTCP: BOOL;
		Robot8_Reqs_TraccTCP: BOOL;
		Robot9_Reqs_TraccTCP: BOOL;
		Robot10_Reqs_TraccTCP: BOOL;
		Robot11_Reqs_TraccTCP: BOOL;
		Robot12_Reqs_TraccTCP: BOOL;
		Robot13_Reqs_TraccTCP: BOOL;
		Robot14_Reqs_TraccTCP: BOOL;
		Robot15_Reqs_TraccTCP: BOOL;
		Robot16_Reqs_TraccTCP: BOOL;
		Robot17_Reqs_TraccTCP: BOOL;
		Robot18_Reqs_TraccTCP: BOOL;
		Robot19_Reqs_TraccTCP: BOOL;
		Robot20_Reqs_TraccTCP: BOOL;
		Robot21_Reqs_TraccTCP: BOOL;
		Robot22_Reqs_TraccTCP: BOOL;
		Robot23_Reqs_TraccTCP: BOOL;
		Robot24_Reqs_TraccTCP: BOOL;
		Robot25_Reqs_TraccTCP: BOOL;
		Robot26_Reqs_TraccTCP: BOOL;
		Robot27_Reqs_TraccTCP: BOOL;
		Robot28_Reqs_TraccTCP: BOOL;
		Robot29_Reqs_TraccTCP: BOOL;
		Robot30_Reqs_TraccTCP: BOOL;
				
		Prod_Inc: R_TRIG;
		Cycle_Time: TON;
		Cycle_Time_Pulse: R_TRIG;
		Date_Stamp_TMR: TON;
		Date_StampHome_TMR: TON;
		CLFaulted:BOOL;
		PPFaulted: BOOL;

(*Non-Standard Variables*)

		(*FB Instances*)
		(*Tool Positions*)
			(*Add User Indivdual Position Variables Here*)

		(*Part Present Sensors*)
			(*Add User Sensor Variables Here*)
		(*Motion Sequence Variables*)
			Clamp_Step: UINT;
			Repo1_Step: UINT;
			Repo2_Step: UINT;
			Repo3_Step: UINT;
			Repo4_Step: UINT;
			Unclamp_Step: UINT;

	END_VAR

	(*data that needs to be retained in the event of a power cycle*)
	VAR PERSISTENT
		Master_Tests_Complete: BOOL;
		Brake_Tests_Complete: BOOL;
		Tip_Change_Complete: BOOL;
		Tip_Dress_CompleteAll:BOOL;
		Tip_Dress_Complete1:BOOL;
		Tip_Dress_Complete2:BOOL;
		Tip_Dress_Complete3:BOOL;
		Tip_Dress_Complete4:BOOL;
		Tip_Dress_Complete5:BOOL;
		Tip_Dress_Complete6:BOOL;
		Tip_Dress_Complete7:BOOL;
		Tip_Dress_Complete8:BOOL;
		Tip_Dress_Complete9:BOOL;
		Tip_Dress_Complete10:BOOL;
		Tip_Dress_Complete11:BOOL;
		Tip_Dress_Complete12:BOOL;
		Tip_Dress_Complete13:BOOL;
		Tip_Dress_Complete14:BOOL;
		Tip_Dress_Complete15:BOOL;
		Tip_Dress_Complete16:BOOL;
		Tip_Dress_Complete17:BOOL;
		Tip_Dress_Complete18:BOOL;
		Tip_Dress_Complete19:BOOL;
		Tip_Dress_Complete20:BOOL;
		Tip_Dress_Complete21:BOOL;
		Tip_Dress_Complete22:BOOL;
		Tip_Dress_Complete23:BOOL;
		Tip_Dress_Complete24:BOOL;
		Tip_Dress_Complete25:BOOL;
		Tip_Dress_Complete26:BOOL;
		Tip_Dress_Complete27:BOOL;
		Tip_Dress_Complete28:BOOL;
		Tip_Dress_Complete29:BOOL;
		Tip_Dress_Complete30:BOOL;
		
		(*Custom for CCB*)
		TraccTCP_CompleteALL:BOOL;
		TraccTCP_Complete1:BOOL;
		TraccTCP_Complete2:BOOL;
		TraccTCP_Complete3:BOOL;
		TraccTCP_Complete4:BOOL;
		TraccTCP_Complete5:BOOL;
		TraccTCP_Complete6:BOOL;
		TraccTCP_Complete7:BOOL;
		TraccTCP_Complete8:BOOL;
		TraccTCP_Complete9:BOOL;
		TraccTCP_Complete10:BOOL;
		TraccTCP_Complete11:BOOL;
		TraccTCP_Complete12:BOOL;
		TraccTCP_Complete13:BOOL;
		TraccTCP_Complete14:BOOL;
		TraccTCP_Complete15:BOOL;
		TraccTCP_Complete16:BOOL;
		TraccTCP_Complete17:BOOL;
		TraccTCP_Complete18:BOOL;
		TraccTCP_Complete19:BOOL;
		TraccTCP_Complete20:BOOL;
		TraccTCP_Complete21:BOOL;
		TraccTCP_Complete22:BOOL;
		TraccTCP_Complete23:BOOL;
		TraccTCP_Complete24:BOOL;
		TraccTCP_Complete25:BOOL;
		TraccTCP_Complete26:BOOL;
		TraccTCP_Complete27:BOOL;
		TraccTCP_Complete28:BOOL;
		TraccTCP_Complete29:BOOL;
		TraccTCP_Complete30:BOOL;

		Cycle_Complete: BOOL;
		Production_Count:INT;
		Repo_REQS: UINT;

		Human_Reqs_MasterTest: BOOL;
		Human_Reqs_BrakeTest: BOOL;
		Human_Reqs_TipChange: BOOL;
		All_RobotsReq_MasterTest: BOOL;
		All_RobotsReq_BrakeTest: BOOL;
		A_Robot_Reqs_MasterTest: BOOL;
		A_Robot_Reqs_BrakeTest: BOOL;
		Robot_Reqs_TipChange: BOOL;
		TipChange_Reqs_TipDress: BOOL;

		Human_Reqs_TipDressR1: BOOL;
		Human_Reqs_TipDressR2: BOOL;
		Human_Reqs_TipDressR3: BOOL;
		Human_Reqs_TipDressR4: BOOL;
		Human_Reqs_TipDressR5: BOOL;
		Human_Reqs_TipDressR6: BOOL;
		Human_Reqs_TipDressR7: BOOL;
		Human_Reqs_TipDressR8: BOOL;
		Human_Reqs_TipDressR9: BOOL;
		Human_Reqs_TipDressR10: BOOL;
		Human_Reqs_TipDressR11: BOOL;
		Human_Reqs_TipDressR12: BOOL;
		Human_Reqs_TipDressR13: BOOL;
		Human_Reqs_TipDressR14: BOOL;
		Human_Reqs_TipDressR15: BOOL;
		Human_Reqs_TipDressR16: BOOL;
		Human_Reqs_TipDressR17: BOOL;
		Human_Reqs_TipDressR18: BOOL;
		Human_Reqs_TipDressR19: BOOL;
		Human_Reqs_TipDressR20: BOOL;
		Human_Reqs_TipDressR21: BOOL;
		Human_Reqs_TipDressR22: BOOL;
		Human_Reqs_TipDressR23: BOOL;
		Human_Reqs_TipDressR24: BOOL;
		Human_Reqs_TipDressR25: BOOL;
		Human_Reqs_TipDressR26: BOOL;
		Human_Reqs_TipDressR27: BOOL;
		Human_Reqs_TipDressR28: BOOL;
		Human_Reqs_TipDressR29: BOOL;
		Human_Reqs_TipDressR30: BOOL;
		
		Human_Reqs_TraccTCP_R1: BOOL;
		Human_Reqs_TraccTCP_R2: BOOL;
		Human_Reqs_TraccTCP_R3: BOOL;
		Human_Reqs_TraccTCP_R4: BOOL;
		Human_Reqs_TraccTCP_R5: BOOL;
		Human_Reqs_TraccTCP_R6: BOOL;
		Human_Reqs_TraccTCP_R7: BOOL;
		Human_Reqs_TraccTCP_R8: BOOL;
		Human_Reqs_TraccTCP_R9: BOOL;
		Human_Reqs_TraccTCP_R10: BOOL;
		Human_Reqs_TraccTCP_R11: BOOL;
		Human_Reqs_TraccTCP_R12: BOOL;
		Human_Reqs_TraccTCP_R13: BOOL;
		Human_Reqs_TraccTCP_R14: BOOL;
		Human_Reqs_TraccTCP_R15: BOOL;
		Human_Reqs_TraccTCP_R16: BOOL;
		Human_Reqs_TraccTCP_R17: BOOL;
		Human_Reqs_TraccTCP_R18: BOOL;
		Human_Reqs_TraccTCP_R19: BOOL;
		Human_Reqs_TraccTCP_R20: BOOL;
		Human_Reqs_TraccTCP_R21: BOOL;
		Human_Reqs_TraccTCP_R22: BOOL;
		Human_Reqs_TraccTCP_R23: BOOL;
		Human_Reqs_TraccTCP_R24: BOOL;
		Human_Reqs_TraccTCP_R25: BOOL;
		Human_Reqs_TraccTCP_R26: BOOL;
		Human_Reqs_TraccTCP_R27: BOOL;
		Human_Reqs_TraccTCP_R28: BOOL;
		Human_Reqs_TraccTCP_R29: BOOL;
		Human_Reqs_TraccTCP_R30: BOOL;
	END_VAR

	VAR_OUTPUT
		Prog_Ok: BOOL;
		Prod_Count_Out: INT;
		Cycle_Time_Out: TIME;
		PrevCycle_Time_Out: TIME;
		Model_ID: UINT;
		Service_Call_ForAllRobots: BOOL;
		Service_Call_ForRobot1: BOOL;
		Service_Call_ForRobot2: BOOL;
		Service_Call_ForRobot3: BOOL;
		Service_Call_ForRobot4: BOOL;
		Service_Call_ForRobot5: BOOL;
		Service_Call_ForRobot6: BOOL;
		Service_Call_ForRobot7: BOOL;
		Service_Call_ForRobot8: BOOL;
		Service_Call_ForRobot9: BOOL;
		Service_Call_ForRobot10: BOOL;
		Service_Call_ForRobot11: BOOL;
		Service_Call_ForRobot12: BOOL;
		Service_Call_ForRobot13: BOOL;
		Service_Call_ForRobot14: BOOL;
		Service_Call_ForRobot15: BOOL;
		Service_Call_ForRobot16: BOOL;
		Service_Call_ForRobot17: BOOL;
		Service_Call_ForRobot18: BOOL;
		Service_Call_ForRobot19: BOOL;
		Service_Call_ForRobot20: BOOL;
		Service_Call_ForRobot21: BOOL;
		Service_Call_ForRobot22: BOOL;
		Service_Call_ForRobot23: BOOL;
		Service_Call_ForRobot24: BOOL;
		Service_Call_ForRobot25: BOOL;
		Service_Call_ForRobot26: BOOL;
		Service_Call_ForRobot27: BOOL;
		Service_Call_ForRobot28: BOOL;
		Service_Call_ForRobot29: BOOL;
		Service_Call_ForRobot30: BOOL;
		Robots_Clear_ToProceed: BOOL;
		Task_ID: UINT;
		Fix_ID: UINT;
		All_Complete_Ack: BOOL;
		Repo_Ack: UINT;
		Rxx_ReadyAt_TipChangePosition: UDINT;
	END_VAR



	(*Set FB_OK to True*)
	Prog_OK:= TRUE;
(*$$$$$$$$$$$$$$$$$$$$$$$$$$$$$$$$$$$$$$$$$$$$$$$$Gather Status Of Hardware $$$$$$$$$$$$$$$$$$$$$$$$$$$$$$$$$$$$$$$$$$$$$$$$$$$$*)
	(*Discrete I/O Node*)

(*$$$$$$$$$$$$$$$$$$$$$$$$$$$$$$$$$$$$$$$$$$$$$$$$$$ Gather Safety Inputs $$$$$$$$$$$$$$$$$$$$$$$$$$$$$$$$$$$$$$$$$$$$$$$$$$$$$$$*)


(*$$$$$$$$$$$$$$$$$$$$$$$$$$$$$$$$$$$$$$$$$$$$$$$$$ Gather Standard Inputs $$$$$$$$$$$$$$$$$$$$$$$$$$$$$$$$$$$$$$$$$$$$$$$$$$$$$$*)
(*Master Test Request from any IC*)
	IF In_From_ICxx.Force_Master_Test
		THEN
			Human_Reqs_MasterTest:= TRUE; (*Reset at Master_Test_Complete*)
	END_IF;
(*Master Test Reqs from any Robot*)
	IF NOT GTAC_CONFIG.Under_Construction
		AND (MAIN.R1.Master_Test_Reqd
			OR MAIN.R2.Master_Test_Reqd
			OR MAIN.R3.Master_Test_Reqd
			OR MAIN.R4.Master_Test_Reqd
			OR MAIN.R5.Master_Test_Reqd
			OR MAIN.R6.Master_Test_Reqd
			OR MAIN.R7.Master_Test_Reqd
			OR MAIN.R8.Master_Test_Reqd
			OR MAIN.R9.Master_Test_Reqd
			OR MAIN.R10.Master_Test_Reqd
			OR MAIN.R11.Master_Test_Reqd
			OR MAIN.R12.Master_Test_Reqd
			OR MAIN.R13.Master_Test_Reqd
			OR MAIN.R14.Master_Test_Reqd
			OR MAIN.R15.Master_Test_Reqd
			OR MAIN.R16.Master_Test_Reqd
			OR MAIN.R17.Master_Test_Reqd
			OR MAIN.R18.Master_Test_Reqd
			OR MAIN.R19.Master_Test_Reqd
			OR MAIN.R20.Master_Test_Reqd
			OR MAIN.R21.Master_Test_Reqd
			OR MAIN.R22.Master_Test_Reqd
			OR MAIN.R23.Master_Test_Reqd
			OR MAIN.R24.Master_Test_Reqd
			OR MAIN.R25.Master_Test_Reqd
			OR MAIN.R26.Master_Test_Reqd
			OR MAIN.R27.Master_Test_Reqd
			OR MAIN.R28.Master_Test_Reqd
			OR MAIN.R29.Master_Test_Reqd
			OR MAIN.R30.Master_Test_Reqd)
	THEN

                   	A_Robot_Reqs_MasterTest := TRUE;  (*Reset at Master Test_Complete*)

	END_IF;



(*Brake Test Request from any IC*)
	IF In_From_ICxx.Force_Brake_Test
		THEN
			Human_Reqs_BrakeTest:= TRUE; (*Reset at Brake_Test_Complete*)
	END_IF;
(*Brake Test Reqs from any Robot*)
	IF NOT GTAC_CONFIG.Under_Construction
 		AND NOT All_RobotsReq_BrakeTest
                    AND (MAIN.R1.Brake_Test_Reqd
				OR MAIN.R2.Brake_Test_Reqd
				OR MAIN.R3.Brake_Test_Reqd
				OR MAIN.R4.Brake_Test_Reqd
				OR MAIN.R5.Brake_Test_Reqd
				OR MAIN.R6.Brake_Test_Reqd
				OR MAIN.R7.Brake_Test_Reqd
				OR MAIN.R8.Brake_Test_Reqd
				OR MAIN.R9.Brake_Test_Reqd
				OR MAIN.R10.Brake_Test_Reqd
				OR MAIN.R11.Brake_Test_Reqd
				OR MAIN.R12.Brake_Test_Reqd
				OR MAIN.R13.Brake_Test_Reqd
				OR MAIN.R14.Brake_Test_Reqd
				OR MAIN.R15.Brake_Test_Reqd
				OR MAIN.R16.Brake_Test_Reqd
				OR MAIN.R17.Brake_Test_Reqd
				OR MAIN.R18.Brake_Test_Reqd
				OR MAIN.R19.Brake_Test_Reqd
				OR MAIN.R20.Brake_Test_Reqd
				OR MAIN.R21.Brake_Test_Reqd
				OR MAIN.R22.Brake_Test_Reqd
				OR MAIN.R23.Brake_Test_Reqd
				OR MAIN.R24.Brake_Test_Reqd
				OR MAIN.R25.Brake_Test_Reqd
				OR MAIN.R26.Brake_Test_Reqd
				OR MAIN.R27.Brake_Test_Reqd
				OR MAIN.R28.Brake_Test_Reqd
				OR MAIN.R29.Brake_Test_Reqd
				OR MAIN.R30.Brake_Test_Reqd)
	THEN

                           		A_Robot_Reqs_BrakeTest := TRUE;  (*Reset at Brake Test_Complete*)

	END_IF;

(*Brake Test Reqs from ALL Robots*)
	IF NOT GTAC_CONFIG.Under_Construction
                     AND (MAIN.R1.Brake_Test_Reqd AND
				(MAIN.R2.Brake_Test_Reqd OR GTAC_CONFIG.Option_Robot_Count<2) AND
				(MAIN.R3.Brake_Test_Reqd OR GTAC_CONFIG.Option_Robot_Count<3) AND
				(MAIN.R4.Brake_Test_Reqd OR GTAC_CONFIG.Option_Robot_Count<4) AND
				(MAIN.R5.Brake_Test_Reqd OR GTAC_CONFIG.Option_Robot_Count<5) AND
				(MAIN.R6.Brake_Test_Reqd OR GTAC_CONFIG.Option_Robot_Count<6) AND
				(MAIN.R7.Brake_Test_Reqd OR GTAC_CONFIG.Option_Robot_Count<7) AND
				(MAIN.R8.Brake_Test_Reqd OR GTAC_CONFIG.Option_Robot_Count<8) AND
				(MAIN.R9.Brake_Test_Reqd OR GTAC_CONFIG.Option_Robot_Count<9) AND
				(MAIN.R10.Brake_Test_Reqd OR GTAC_CONFIG.Option_Robot_Count<10) AND
				(MAIN.R11.Brake_Test_Reqd OR GTAC_CONFIG.Option_Robot_Count<11) AND
				(MAIN.R12.Brake_Test_Reqd OR GTAC_CONFIG.Option_Robot_Count<12) AND
				(MAIN.R13.Brake_Test_Reqd OR GTAC_CONFIG.Option_Robot_Count<13) AND
				(MAIN.R14.Brake_Test_Reqd OR GTAC_CONFIG.Option_Robot_Count<14) AND
				(MAIN.R15.Brake_Test_Reqd OR GTAC_CONFIG.Option_Robot_Count<15) AND
				(MAIN.R16.Brake_Test_Reqd OR GTAC_CONFIG.Option_Robot_Count<16) AND
				(MAIN.R17.Brake_Test_Reqd OR GTAC_CONFIG.Option_Robot_Count<17) AND
				(MAIN.R18.Brake_Test_Reqd OR GTAC_CONFIG.Option_Robot_Count<18) AND
				(MAIN.R19.Brake_Test_Reqd OR GTAC_CONFIG.Option_Robot_Count<19) AND
				(MAIN.R20.Brake_Test_Reqd OR GTAC_CONFIG.Option_Robot_Count<20) AND
				(MAIN.R21.Brake_Test_Reqd OR GTAC_CONFIG.Option_Robot_Count<21) AND
				(MAIN.R22.Brake_Test_Reqd OR GTAC_CONFIG.Option_Robot_Count<22) AND
				(MAIN.R23.Brake_Test_Reqd OR GTAC_CONFIG.Option_Robot_Count<23) AND
				(MAIN.R24.Brake_Test_Reqd OR GTAC_CONFIG.Option_Robot_Count<24) AND
				(MAIN.R25.Brake_Test_Reqd OR GTAC_CONFIG.Option_Robot_Count<25) AND
				(MAIN.R26.Brake_Test_Reqd OR GTAC_CONFIG.Option_Robot_Count<26) AND
				(MAIN.R27.Brake_Test_Reqd OR GTAC_CONFIG.Option_Robot_Count<27) AND
				(MAIN.R28.Brake_Test_Reqd OR GTAC_CONFIG.Option_Robot_Count<28) AND
				(MAIN.R29.Brake_Test_Reqd OR GTAC_CONFIG.Option_Robot_Count<29) AND
				(MAIN.R30.Brake_Test_Reqd OR GTAC_CONFIG.Option_Robot_Count<30))
	THEN

                           		All_RobotsReq_BrakeTest := TRUE;  (*Reset at Brake Test_Complete*)
				A_Robot_Reqs_BrakeTest := FALSE;
				Human_Reqs_BrakeTest:= FALSE;

	END_IF;


(*TipChange Request from any IC*)
	IF In_From_ICxx.Force_TipChange
		THEN
			Human_Reqs_TipChange:= TRUE; (*Reset at Tip_Change_Complete*)
	END_IF;

(*Tip Change Requests from any Robot (WCU)*)
  	IF NOT GTAC_CONFIG.Under_Construction
                     	AND ((MAIN.R1.Any_WCU_TipChng_Rqst) OR (MAIN.R2.Any_WCU_TipChng_Rqst) OR (MAIN.R3.Any_WCU_TipChng_Rqst)
                                	OR (MAIN.R4.Any_WCU_TipChng_Rqst) OR (MAIN.R5.Any_WCU_TipChng_Rqst)	OR (MAIN.R6.Any_WCU_TipChng_Rqst)
                                	OR (MAIN.R7.Any_WCU_TipChng_Rqst) OR (MAIN.R8.Any_WCU_TipChng_Rqst) OR (MAIN.R9.Any_WCU_TipChng_Rqst)
                                	OR (MAIN.R10.Any_WCU_TipChng_Rqst) OR (MAIN.R11.Any_WCU_TipChng_Rqst) OR (MAIN.R12.Any_WCU_TipChng_Rqst)
                                	OR (MAIN.R13.Any_WCU_TipChng_Rqst) OR (MAIN.R14.Any_WCU_TipChng_Rqst) OR (MAIN.R15.Any_WCU_TipChng_Rqst)
                                	OR (MAIN.R16.Any_WCU_TipChng_Rqst) OR (MAIN.R17.Any_WCU_TipChng_Rqst) OR (MAIN.R18.Any_WCU_TipChng_Rqst)
                                	OR (MAIN.R19.Any_WCU_TipChng_Rqst) OR (MAIN.R20.Any_WCU_TipChng_Rqst) OR (MAIN.R21.Any_WCU_TipChng_Rqst)
                                	OR (MAIN.R22.Any_WCU_TipChng_Rqst) OR (MAIN.R23.Any_WCU_TipChng_Rqst) OR (MAIN.R24.Any_WCU_TipChng_Rqst)
                                	OR (MAIN.R25.Any_WCU_TipChng_Rqst) OR (MAIN.R26.Any_WCU_TipChng_Rqst) OR (MAIN.R27.Any_WCU_TipChng_Rqst)
                                	OR (MAIN.R28.Any_WCU_TipChng_Rqst) OR (MAIN.R29.Any_WCU_TipChng_Rqst) OR (MAIN.R30.Any_WCU_TipChng_Rqst))
						OR In_From_ICxx.Force_TipChange
	THEN

                                                                Robot_Reqs_TipChange := TRUE;  (*Reset at Tip_Change_Complete*)

	END_IF;

(*All Steppers Are Reset*)
All_Robots_SteppersRST:= (MAIN.R1.All_WCUSteppers_Reset AND
						(MAIN.R2.All_WCUSteppers_Reset OR GTAC_CONFIG.Option_Robot_Count<2) AND
						(MAIN.R3.All_WCUSteppers_Reset OR GTAC_CONFIG.Option_Robot_Count<3) AND
						(MAIN.R4.All_WCUSteppers_Reset OR GTAC_CONFIG.Option_Robot_Count<4) AND
						(MAIN.R5.All_WCUSteppers_Reset OR GTAC_CONFIG.Option_Robot_Count<5) AND
						(MAIN.R6.All_WCUSteppers_Reset OR GTAC_CONFIG.Option_Robot_Count<6) AND
						(MAIN.R7.All_WCUSteppers_Reset OR GTAC_CONFIG.Option_Robot_Count<7) AND
						(MAIN.R8.All_WCUSteppers_Reset OR GTAC_CONFIG.Option_Robot_Count<8) AND
						(MAIN.R9.All_WCUSteppers_Reset OR GTAC_CONFIG.Option_Robot_Count<9) AND
						(MAIN.R10.All_WCUSteppers_Reset OR GTAC_CONFIG.Option_Robot_Count<10) AND
						(MAIN.R11.All_WCUSteppers_Reset OR GTAC_CONFIG.Option_Robot_Count<11) AND
						(MAIN.R12.All_WCUSteppers_Reset OR GTAC_CONFIG.Option_Robot_Count<12) AND
						(MAIN.R13.All_WCUSteppers_Reset OR GTAC_CONFIG.Option_Robot_Count<13) AND
						(MAIN.R14.All_WCUSteppers_Reset OR GTAC_CONFIG.Option_Robot_Count<14) AND
						(MAIN.R15.All_WCUSteppers_Reset OR GTAC_CONFIG.Option_Robot_Count<15) AND
						(MAIN.R16.All_WCUSteppers_Reset OR GTAC_CONFIG.Option_Robot_Count<16) AND
						(MAIN.R17.All_WCUSteppers_Reset OR GTAC_CONFIG.Option_Robot_Count<17) AND
						(MAIN.R18.All_WCUSteppers_Reset OR GTAC_CONFIG.Option_Robot_Count<18) AND
						(MAIN.R19.All_WCUSteppers_Reset OR GTAC_CONFIG.Option_Robot_Count<19) AND
						(MAIN.R20.All_WCUSteppers_Reset OR GTAC_CONFIG.Option_Robot_Count<20) AND
						(MAIN.R21.All_WCUSteppers_Reset OR GTAC_CONFIG.Option_Robot_Count<21) AND
						(MAIN.R22.All_WCUSteppers_Reset OR GTAC_CONFIG.Option_Robot_Count<22) AND
						(MAIN.R23.All_WCUSteppers_Reset OR GTAC_CONFIG.Option_Robot_Count<23) AND
						(MAIN.R24.All_WCUSteppers_Reset OR GTAC_CONFIG.Option_Robot_Count<24) AND
						(MAIN.R25.All_WCUSteppers_Reset OR GTAC_CONFIG.Option_Robot_Count<25) AND
						(MAIN.R26.All_WCUSteppers_Reset OR GTAC_CONFIG.Option_Robot_Count<26) AND
						(MAIN.R27.All_WCUSteppers_Reset OR GTAC_CONFIG.Option_Robot_Count<27) AND
						(MAIN.R28.All_WCUSteppers_Reset OR GTAC_CONFIG.Option_Robot_Count<28) AND
						(MAIN.R29.All_WCUSteppers_Reset OR GTAC_CONFIG.Option_Robot_Count<29) AND
						(MAIN.R30.All_WCUSteppers_Reset OR GTAC_CONFIG.Option_Robot_Count<30))
						OR GTAC_CONFIG.Under_Construction;

(*Tip Dress Request Section*)
(*TipDress Request from any IC*)
IF In_From_ICxx.R1_Dress_Req
	THEN
		Human_Reqs_TipDressR1:= TRUE; (*Reset at Tip_Dress_Complete1*)
END_IF;
(*Tip Dress/Ream Requests from Robots (WCU)*)
(*Robot #1 Tip Dress Request*)
IF (MAIN.R1.WCU1_DressReqd_1
	OR MAIN.R1.WCU1_DressReqd_2
	OR MAIN.R1.Ream_Reqd)
	THEN
		Robot1_Reqs_TipDress:= TRUE;
END_IF;

(*TipDress Request from any IC*)
IF In_From_ICxx.R2_Dress_Req
	THEN
		Human_Reqs_TipDressR2:= TRUE; (*Reset at Tip_Dress_Complete2*)
END_IF;
(*Robot #2 Tip Dress Request*)
IF (MAIN.R2.WCU1_DressReqd_1
	OR MAIN.R2.WCU1_DressReqd_2
	OR MAIN.R2.Ream_Reqd)
	THEN
		Robot2_Reqs_TipDress:= TRUE;
END_IF;

(*TipDress Request from any IC*)
IF In_From_ICxx.R3_Dress_Req
	THEN
		Human_Reqs_TipDressR3:= TRUE; (*Reset at Tip_Dress_Complete3*)
END_IF;
(*Robot #3 Tip Dress Request*)
IF (MAIN.R3.WCU1_DressReqd_1
	OR MAIN.R3.WCU1_DressReqd_2
	OR MAIN.R3.Ream_Reqd)
	THEN
		Robot3_Reqs_TipDress:= TRUE;
END_IF;

(*TipDress Request from any IC*)
IF In_From_ICxx.R4_Dress_Req
	THEN
		Human_Reqs_TipDressR4:= TRUE; (*Reset at Tip_Dress_Complete4*)
END_IF;
(*Robot #4 Tip Dress Request*)
IF (MAIN.R4.WCU1_DressReqd_1
	OR MAIN.R4.WCU1_DressReqd_2
	OR MAIN.R4.Ream_Reqd)
	THEN
		Robot4_Reqs_TipDress:=TRUE;
END_IF;

(*TipDress Request from any IC*)
IF In_From_ICxx.R5_Dress_Req
	THEN
		Human_Reqs_TipDressR5:= TRUE; (*Reset at Tip_Dress_Complete5*)
END_IF;
(*Robot #5 Tip Dress Request*)
IF (MAIN.R5.WCU1_DressReqd_1
	OR MAIN.R5.WCU1_DressReqd_2
	OR MAIN.R5.Ream_Reqd)
	THEN
		Robot5_Reqs_TipDress:= TRUE;
END_IF;

(*TipDress Request from any IC*)
IF In_From_ICxx.R6_Dress_Req
	THEN
		Human_Reqs_TipDressR6:= TRUE; (*Reset at Tip_Dress_Complete6*)
END_IF;
(*Robot #6 Tip Dress Request*)
IF (MAIN.R6.WCU1_DressReqd_1
	OR MAIN.R6.WCU1_DressReqd_2
	OR MAIN.R6.Ream_Reqd)
	THEN
		Robot6_Reqs_TipDress:= TRUE;
END_IF;

(*TipDress Request from any IC*)
IF In_From_ICxx.R7_Dress_Req
	THEN
		Human_Reqs_TipDressR7:= TRUE; (*Reset at Tip_Dress_Complete7*)
END_IF;
(*Robot #7 Tip Dress Request*)
IF (MAIN.R7.WCU1_DressReqd_1
	OR MAIN.R7.WCU1_DressReqd_2
	OR MAIN.R7.Ream_Reqd)
	THEN
		Robot7_Reqs_TipDress:= TRUE;
END_IF;

(*TipDress Request from any IC*)
IF In_From_ICxx.R8_Dress_Req
	THEN
		Human_Reqs_TipDressR8:= TRUE; (*Reset at Tip_Dress_Complete8*)
END_IF;
(*Robot #8 Tip Dress Request*)
IF (MAIN.R8.WCU1_DressReqd_1
	OR MAIN.R8.WCU1_DressReqd_2
	OR MAIN.R8.Ream_Reqd)
	THEN
		Robot8_Reqs_TipDress:= TRUE;
END_IF;

(*TipDress Request from any IC*)
IF In_From_ICxx.R9_Dress_Req
	THEN
		Human_Reqs_TipDressR9:= TRUE; (*Reset at Tip_Dress_Complete9*)
END_IF;
(*Robot #9 Tip Dress Request*)
IF (MAIN.R9.WCU1_DressReqd_1
	OR MAIN.R9.WCU1_DressReqd_2
	OR MAIN.R9.Ream_Reqd)
	THEN
		Robot9_Reqs_TipDress:= TRUE;
END_IF;

(*TipDress Request from any IC*)
IF In_From_ICxx.R10_Dress_Req
	THEN
		Human_Reqs_TipDressR10:= TRUE; (*Reset at Tip_Dress_Complete10*)
END_IF;
(*Robot #10 Tip Dress Request*)
IF (MAIN.R10.WCU1_DressReqd_1
	OR MAIN.R10.WCU1_DressReqd_2
	OR MAIN.R10.Ream_Reqd)
	THEN
		Robot10_Reqs_TipDress:= TRUE;
END_IF;

(*TipDress Request from any IC*)
IF In_From_ICxx.R11_Dress_Req
	THEN
		Human_Reqs_TipDressR11:= TRUE; (*Reset at Tip_Dress_Complete11*)
END_IF;
(*Robot #11 Tip Dress Request*)
IF (MAIN.R11.WCU1_DressReqd_1
	OR MAIN.R11.WCU1_DressReqd_2
	OR MAIN.R11.Ream_Reqd)
	THEN
		Robot11_Reqs_TipDress:= TRUE;
END_IF;

(*TipDress Request from any IC*)
IF In_From_ICxx.R12_Dress_Req
	THEN
		Human_Reqs_TipDressR12:= TRUE; (*Reset at Tip_Dress_Complete12*)
END_IF;
(*Robot #12 Tip Dress Request*)
IF (MAIN.R12.WCU1_DressReqd_1
	OR MAIN.R12.WCU1_DressReqd_2
	OR MAIN.R12.Ream_Reqd)
	THEN
		Robot12_Reqs_TipDress:= TRUE;
END_IF;

(*TipDress Request from any IC*)
IF In_From_ICxx.R13_Dress_Req
	THEN
		Human_Reqs_TipDressR13:= TRUE; (*Reset at Tip_Dress_Complete13*)
END_IF;
(*Robot #13 Tip Dress Request*)
IF (MAIN.R13.WCU1_DressReqd_1
	OR MAIN.R13.WCU1_DressReqd_2
	OR MAIN.R13.Ream_Reqd)
	THEN
		Robot13_Reqs_TipDress:=TRUE;
END_IF;

(*TipDress Request from any IC*)
IF In_From_ICxx.R14_Dress_Req
	THEN
		Human_Reqs_TipDressR14:= TRUE; (*Reset at Tip_Dress_Complete14*)
END_IF;
(*Robot #14 Tip Dress Request*)
IF (MAIN.R14.WCU1_DressReqd_1
	OR MAIN.R14.WCU1_DressReqd_2
	OR MAIN.R14.Ream_Reqd)
	THEN
		Robot14_Reqs_TipDress:= TRUE;
END_IF;

(*TipDress Request from any IC*)
IF In_From_ICxx.R15_Dress_Req
	THEN
		Human_Reqs_TipDressR15:= TRUE; (*Reset at Tip_Dress_Complete15*)
END_IF;
(*Robot #15 Tip Dress Request*)
IF (MAIN.R15.WCU1_DressReqd_1
	OR MAIN.R15.WCU1_DressReqd_2
	OR MAIN.R15.Ream_Reqd)
	THEN
		Robot15_Reqs_TipDress:= TRUE;
END_IF;

(*TipDress Request from any IC*)
IF In_From_ICxx.R16_Dress_Req
	THEN
		Human_Reqs_TipDressR16:= TRUE; (*Reset at Tip_Dress_Complete16*)
END_IF;
(*Robot #16 Tip Dress Request*)
IF (MAIN.R16.WCU1_DressReqd_1
	OR MAIN.R16.WCU1_DressReqd_2
	OR MAIN.R16.Ream_Reqd)
	THEN
		Robot16_Reqs_TipDress:= TRUE;
END_IF;

(*TipDress Request from any IC*)
IF In_From_ICxx.R17_Dress_Req
	THEN
		Human_Reqs_TipDressR17:= TRUE; (*Reset at Tip_Dress_Complete17*)
END_IF;
(*Robot #17 Tip Dress Request*)
IF (MAIN.R17.WCU1_DressReqd_1
	OR MAIN.R17.WCU1_DressReqd_2
	OR MAIN.R17.Ream_Reqd)
	THEN
		Robot17_Reqs_TipDress:= TRUE;
END_IF;

(*TipDress Request from any IC*)
IF In_From_ICxx.R18_Dress_Req
	THEN
		Human_Reqs_TipDressR18:= TRUE; (*Reset at Tip_Dress_Complete18*)
END_IF;
(*Robot #18 Tip Dress Request*)
IF (MAIN.R18.WCU1_DressReqd_1
	OR MAIN.R18.WCU1_DressReqd_2
	OR MAIN.R18.Ream_Reqd)
	THEN
		Robot18_Reqs_TipDress:= TRUE;
END_IF;

(*TipDress Request from any IC*)
IF In_From_ICxx.R19_Dress_Req
	THEN
		Human_Reqs_TipDressR19:= TRUE; (*Reset at Tip_Dress_Complete19*)
END_IF;
(*Robot #19 Tip Dress Request*)
IF (MAIN.R19.WCU1_DressReqd_1
	OR MAIN.R19.WCU1_DressReqd_2
	OR MAIN.R19.Ream_Reqd)
	THEN
		Robot19_Reqs_TipDress:= TRUE;
END_IF;

(*TipDress Request from any IC*)
IF In_From_ICxx.R20_Dress_Req
	THEN
		Human_Reqs_TipDressR20:= TRUE; (*Reset at Tip_Dress_Complete20*)
END_IF;
(*Robot #20 Tip Dress Request*)
IF (MAIN.R20.WCU1_DressReqd_1
	OR MAIN.R20.WCU1_DressReqd_2
	OR MAIN.R20.Ream_Reqd)
	THEN
		Robot20_Reqs_TipDress:= TRUE;
END_IF;

(*TipDress Request from any IC*)
IF In_From_ICxx.R21_Dress_Req
	THEN
		Human_Reqs_TipDressR21:= TRUE; (*Reset at Tip_Dress_Complete21*)
END_IF;
(*Robot #21 Tip Dress Request*)
IF (MAIN.R21.WCU1_DressReqd_1
	OR MAIN.R21.WCU1_DressReqd_2
	OR MAIN.R21.Ream_Reqd)
	THEN
		Robot21_Reqs_TipDress:= TRUE;
END_IF;

(*TipDress Request from any IC*)
IF In_From_ICxx.R22_Dress_Req
	THEN
		Human_Reqs_TipDressR22:= TRUE; (*Reset at Tip_Dress_Complete22*)
END_IF;
(*Robot #22 Tip Dress Request*)
IF (MAIN.R22.WCU1_DressReqd_1 OR MAIN.R22.WCU1_DressReqd_2)
	THEN
		Robot22_Reqs_TipDress:= TRUE;
END_IF;

(*TipDress Request from any IC*)
IF In_From_ICxx.R23_Dress_Req
	THEN
		Human_Reqs_TipDressR23:= TRUE; (*Reset at Tip_Dress_Complete23*)
END_IF;
(*Robot #23 Tip Dress Request*)
IF (MAIN.R23.WCU1_DressReqd_1
	OR MAIN.R23.WCU1_DressReqd_2
	OR MAIN.R23.Ream_Reqd)
	THEN
		Robot23_Reqs_TipDress:= TRUE;
END_IF;

(*TipDress Request from any IC*)
IF In_From_ICxx.R24_Dress_Req
	THEN
		Human_Reqs_TipDressR24:= TRUE; (*Reset at Tip_Dress_Complete24*)
END_IF;
(*Robot #24 Tip Dress Request*)
IF (MAIN.R24.WCU1_DressReqd_1
	OR MAIN.R24.WCU1_DressReqd_2
	OR MAIN.R24.Ream_Reqd)
	THEN
		Robot24_Reqs_TipDress:= TRUE;
END_IF;

(*TipDress Request from any IC*)
IF In_From_ICxx.R25_Dress_Req
	THEN
		Human_Reqs_TipDressR25:= TRUE; (*Reset at Tip_Dress_Complete25*)
END_IF;
(*Robot #25 Tip Dress Request*)
IF (MAIN.R25.WCU1_DressReqd_1
	OR MAIN.R25.WCU1_DressReqd_2
	OR MAIN.R25.Ream_Reqd)
	THEN
		Robot25_Reqs_TipDress:= TRUE;
END_IF;

(*TipDress Request from any IC*)
IF In_From_ICxx.R26_Dress_Req
	THEN
		Human_Reqs_TipDressR26:= TRUE; (*Reset at Tip_Dress_Complete26*)
END_IF;
(*Robot #26 Tip Dress Request*)
IF (MAIN.R26.WCU1_DressReqd_1
	OR MAIN.R26.WCU1_DressReqd_2
	OR MAIN.R26.Ream_Reqd)
	THEN
		Robot26_Reqs_TipDress:= TRUE;
END_IF;

(*TipDress Request from any IC*)
IF In_From_ICxx.R27_Dress_Req
	THEN
		Human_Reqs_TipDressR27:= TRUE; (*Reset at Tip_Dress_Complete27*)
END_IF;
(*Robot #27 Tip Dress Request*)
IF (MAIN.R27.WCU1_DressReqd_1
	OR MAIN.R27.WCU1_DressReqd_2
	OR MAIN.R27.Ream_Reqd)
	THEN
		Robot27_Reqs_TipDress:= TRUE;
END_IF;

(*TipDress Request from any IC*)
IF In_From_ICxx.R28_Dress_Req
	THEN
		Human_Reqs_TipDressR28:= TRUE; (*Reset at Tip_Dress_Complete28*)
END_IF;
(*Robot #28 Tip Dress Request*)
IF (MAIN.R28.WCU1_DressReqd_1
	OR MAIN.R28.WCU1_DressReqd_2
	OR MAIN.R28.Ream_Reqd)
	THEN
		Robot28_Reqs_TipDress:= TRUE;
END_IF;

(*TipDress Request from any IC*)
IF In_From_ICxx.R29_Dress_Req
	THEN
		Human_Reqs_TipDressR29:= TRUE; (*Reset at Tip_Dress_Complete29*)
END_IF;
(*Robot #29 Tip Dress Request*)
IF (MAIN.R29.WCU1_DressReqd_1
	OR MAIN.R29.WCU1_DressReqd_2
	OR MAIN.R29.Ream_Reqd)
	THEN
		Robot29_Reqs_TipDress:= TRUE;
END_IF;

(*TipDress Request from any IC*)
IF In_From_ICxx.R30_Dress_Req
	THEN
		Human_Reqs_TipDressR30:= TRUE; (*Reset at Tip_Dress_Complete30*)
END_IF;
(*Robot #30 Tip Dress Request*)
IF (MAIN.R30.WCU1_DressReqd_1
	OR MAIN.R30.WCU1_DressReqd_2
	OR MAIN.R30.Ream_Reqd)
	THEN
		Robot30_Reqs_TipDress:= TRUE;
END_IF;

(*Gather REQS*)	
	IF Robot1_Reqs_TipDress
		OR Robot2_Reqs_TipDress
		OR Robot3_Reqs_TipDress
		OR Robot4_Reqs_TipDress
		OR Robot5_Reqs_TipDress
		OR Robot6_Reqs_TipDress
		OR Robot7_Reqs_TipDress
		OR Robot8_Reqs_TipDress
		OR Robot9_Reqs_TipDress
		OR Robot10_Reqs_TipDress
		OR Robot11_Reqs_TipDress
		OR Robot12_Reqs_TipDress
		OR Robot13_Reqs_TipDress
		OR Robot14_Reqs_TipDress
		OR Robot15_Reqs_TipDress
		OR Robot16_Reqs_TipDress
		OR Robot17_Reqs_TipDress
		OR Robot18_Reqs_TipDress
		OR Robot19_Reqs_TipDress
		OR Robot20_Reqs_TipDress
		OR Robot21_Reqs_TipDress
		OR Robot22_Reqs_TipDress
		OR Robot23_Reqs_TipDress
		OR Robot24_Reqs_TipDress
		OR Robot25_Reqs_TipDress
		OR Robot26_Reqs_TipDress
		OR Robot27_Reqs_TipDress
		OR Robot28_Reqs_TipDress
		OR Robot29_Reqs_TipDress
		OR Robot30_Reqs_TipDress
		OR In_From_ICxx.Rxx_Dress_Req (*Tip Dress All from UI*)

	THEN
		Robot_Reqs_TipDress:= TRUE;

	END_IF


(*Tracc TCP Requests*)	

(*Robot 1 TraccTCP Request from IC01*)
	IF In_From_ICxx.R1_TraccTCP_Req
		THEN
			Human_Reqs_TraccTCP_R1:= TRUE;		(*Reset at TraccTCP Complete*)
	END_IF
(*Robot 1 TraccTCP Request*)
	IF MAIN.R1.TraccTCP_Reqd
		THEN
			Robot1_Reqs_TraccTCP:= TRUE;
	END_IF
	
(*Robot 2 TraccTCP Request from IC01*)
	IF In_From_ICxx.R2_TraccTCP_Req
		THEN
			Human_Reqs_TraccTCP_R2:= TRUE;		(*Reset at TraccTCP Complete*)
	END_IF
(*Robot 2 TraccTCP Request*)
	IF MAIN.R2.TraccTCP_Reqd
		THEN
			Robot2_Reqs_TraccTCP:= TRUE;
	END_IF
	
(*Robot 3 TraccTCP Request from IC01*)
	IF In_From_ICxx.R3_TraccTCP_Req
		THEN
			Human_Reqs_TraccTCP_R3:= TRUE;		(*Reset at TraccTCP Complete*)
	END_IF
(*Robot 3 TraccTCP Request*)
	IF MAIN.R3.TraccTCP_Reqd
		THEN
			Robot3_Reqs_TraccTCP:= TRUE;
	END_IF;
	
(*Robot 4 TraccTCP Request from IC01*)
	IF In_From_ICxx.R4_TraccTCP_Req
		THEN
			Human_Reqs_TraccTCP_R4:= TRUE;		(*Reset at TraccTCP Complete*)
	END_IF;
(*Robot 4 TraccTCP Request*)
	IF MAIN.R4.TraccTCP_Reqd
		THEN
			Robot4_Reqs_TraccTCP:= TRUE;
	END_IF;

(*Robot 5 TraccTCP Request from IC01*)
	IF In_From_ICxx.R5_TraccTCP_Req
		THEN
			Human_Reqs_TraccTCP_R5:= TRUE;		(*Reset at TraccTCP Complete*)
	END_IF
(*Robot 1 TraccTCP Request*)
	IF MAIN.R5.TraccTCP_Reqd
		THEN
			Robot5_Reqs_TraccTCP:= TRUE;
	END_IF;
	
(*Robot 6 TraccTCP Request from IC01*)
	IF In_From_ICxx.R6_TraccTCP_Req
		THEN
			Human_Reqs_TraccTCP_R6:= TRUE;		(*Reset at TraccTCP Complete*)
	END_IF
(*Robot 6 TraccTCP Request*)
	IF MAIN.R6.TraccTCP_Reqd
		THEN
			Robot6_Reqs_TraccTCP:= TRUE;
	END_IF;
	
(*Robot 7 TraccTCP Request from IC01*)
	IF In_From_ICxx.R7_TraccTCP_Req
		THEN
			Human_Reqs_TraccTCP_R7:= TRUE;		(*Reset at TraccTCP Complete*)
	END_IF;
(*Robot 7 TraccTCP Request*)
	IF MAIN.R7.TraccTCP_Reqd
		THEN
			Robot7_Reqs_TraccTCP:= TRUE;
	END_IF;

(*Robot 8 TraccTCP Request from IC01*)
	IF In_From_ICxx.R8_TraccTCP_Req
		THEN
			Human_Reqs_TraccTCP_R8:= TRUE;		(*Reset at TraccTCP Complete*)
	END_IF;
(*Robot 8 TraccTCP Request*)
	IF MAIN.R8.TraccTCP_Reqd
		THEN
			Robot8_Reqs_TraccTCP:= TRUE;
	END_IF;

(*Robot 9 TraccTCP Request from IC01*)
	IF In_From_ICxx.R9_TraccTCP_Req
		THEN
			Human_Reqs_TraccTCP_R9:= TRUE;		(*Reset at TraccTCP Complete*)
	END_IF;
(*Robot 9 TraccTCP Request*)
	IF MAIN.R9.TraccTCP_Reqd
		THEN
			Robot9_Reqs_TraccTCP:= TRUE;
	END_IF;
	
(*Robot 10 TraccTCP Request from IC01*)
	IF In_From_ICxx.R10_TraccTCP_Req
		THEN
			Human_Reqs_TraccTCP_R10:= TRUE;		(*Reset at TraccTCP Complete*)
	END_IF;
(*Robot 10 TraccTCP Request*)
	IF MAIN.R10.TraccTCP_Reqd
		THEN
			Robot10_Reqs_TraccTCP:= TRUE;
	END_IF;

(*Robot 11 TraccTCP Request from IC01*)
	IF In_From_ICxx.R11_TraccTCP_Req
		THEN
			Human_Reqs_TraccTCP_R11:= TRUE;		(*Reset at TraccTCP Complete*)
	END_IF;
(*Robot 11 TraccTCP Request*)
	IF MAIN.R11.TraccTCP_Reqd
		THEN
			Robot11_Reqs_TraccTCP:= TRUE;
	END_IF;
	
(*Robot 12 TraccTCP Request from IC01*)
	IF In_From_ICxx.R12_TraccTCP_Req
		THEN
			Human_Reqs_TraccTCP_R12:= TRUE;		(*Reset at TraccTCP Complete*)
	END_IF;
(*Robot 12 TraccTCP Request*)
	IF MAIN.R12.TraccTCP_Reqd
		THEN
			Robot12_Reqs_TraccTCP:= TRUE;
	END_IF;
	
(*Robot 13 TraccTCP Request from IC01*)
	IF In_From_ICxx.R13_TraccTCP_Req
		THEN
			Human_Reqs_TraccTCP_R13:= TRUE;		(*Reset at TraccTCP Complete*)
	END_IF;
(*Robot 13 TraccTCP Request*)
	IF MAIN.R13.TraccTCP_Reqd
		THEN
			Robot13_Reqs_TraccTCP:= TRUE;
	END_IF;
	
(*Robot 14 TraccTCP Request from IC01*)
	IF In_From_ICxx.R14_TraccTCP_Req
		THEN
			Human_Reqs_TraccTCP_R14:= TRUE;		(*Reset at TraccTCP Complete*)
	END_IF;
(*Robot 14 TraccTCP Request*)
	IF MAIN.R14.TraccTCP_Reqd
		THEN
			Robot14_Reqs_TraccTCP:= TRUE;
	END_IF;

(*Robot 15 TraccTCP Request from IC01*)
	IF In_From_ICxx.R15_TraccTCP_Req
		THEN
			Human_Reqs_TraccTCP_R15:= TRUE;		(*Reset at TraccTCP Complete*)
	END_IF;
(*Robot 15 TraccTCP Request*)
	IF MAIN.R15.TraccTCP_Reqd
		THEN
			Robot15_Reqs_TraccTCP:= TRUE;
	END_IF;
	
(*Robot 16 TraccTCP Request from IC01*)
	IF In_From_ICxx.R16_TraccTCP_Req
		THEN
			Human_Reqs_TraccTCP_R16:= TRUE;		(*Reset at TraccTCP Complete*)
	END_IF;
(*Robot 16 TraccTCP Request*)
	IF MAIN.R16.TraccTCP_Reqd
		THEN
			Robot16_Reqs_TraccTCP:= TRUE;
	END_IF;
	
(*Robot 17 TraccTCP Request from IC01*)
	IF In_From_ICxx.R17_TraccTCP_Req
		THEN
			Human_Reqs_TraccTCP_R17:= TRUE;		(*Reset at TraccTCP Complete*)
	END_IF;
(*Robot 17 TraccTCP Request*)
	IF MAIN.R17.TraccTCP_Reqd
		THEN
			Robot17_Reqs_TraccTCP:= TRUE;
	END_IF;
	
(*Robot 18 TraccTCP Request from IC01*)
	IF In_From_ICxx.R18_TraccTCP_Req
		THEN
			Human_Reqs_TraccTCP_R18:= TRUE;		(*Reset at TraccTCP Complete*)
	END_IF;
(*Robot 18 TraccTCP Request*)
	IF MAIN.R18.TraccTCP_Reqd
		THEN
			Robot18_Reqs_TraccTCP:= TRUE;
	END_IF;
	
(*Robot 19 TraccTCP Request from IC01*)
	IF In_From_ICxx.R19_TraccTCP_Req
		THEN
			Human_Reqs_TraccTCP_R19:= TRUE;		(*Reset at TraccTCP Complete*)
	END_IF;
(*Robot 19 TraccTCP Request*)
	IF MAIN.R19.TraccTCP_Reqd
		THEN
			Robot19_Reqs_TraccTCP:= TRUE;
	END_IF;
	
(*Robot 20 TraccTCP Request from IC01*)
	IF In_From_ICxx.R20_TraccTCP_Req
		THEN
			Human_Reqs_TraccTCP_R20:= TRUE;		(*Reset at TraccTCP Complete*)
	END_IF;
(*Robot 21 TraccTCP Request*)
	IF MAIN.R21.TraccTCP_Reqd
		THEN
			Robot21_Reqs_TraccTCP:= TRUE;
	END_IF;

(*Robot 21 TraccTCP Request from IC01*)
	IF In_From_ICxx.R21_TraccTCP_Req
		THEN
			Human_Reqs_TraccTCP_R21:= TRUE;		(*Reset at TraccTCP Complete*)
	END_IF;
(*Robot 21 TraccTCP Request*)
	IF MAIN.R21.TraccTCP_Reqd
		THEN
			Robot21_Reqs_TraccTCP:= TRUE;
	END_IF;
	
(*Robot 22 TraccTCP Request from IC01*)
	IF In_From_ICxx.R22_TraccTCP_Req
		THEN
			Human_Reqs_TraccTCP_R22:= TRUE;		(*Reset at TraccTCP Complete*)
	END_IF;
(*Robot 22 TraccTCP Request*)
	IF MAIN.R22.TraccTCP_Reqd
		THEN
			Robot22_Reqs_TraccTCP:= TRUE;
	END_IF;
	
(*Robot 23 TraccTCP Request from IC01*)
	IF In_From_ICxx.R23_TraccTCP_Req
		THEN
			Human_Reqs_TraccTCP_R23:= TRUE;		(*Reset at TraccTCP Complete*)
	END_IF;
(*Robot 23 TraccTCP Request*)
	IF MAIN.R23.TraccTCP_Reqd
		THEN
			Robot23_Reqs_TraccTCP:= TRUE;
	END_IF;
	
(*Robot 24 TraccTCP Request from IC01*)
	IF In_From_ICxx.R24_TraccTCP_Req
		THEN
			Human_Reqs_TraccTCP_R24:= TRUE;		(*Reset at TraccTCP Complete*)
	END_IF;
(*Robot 24 TraccTCP Request*)
	IF MAIN.R24.TraccTCP_Reqd
		THEN
			Robot24_Reqs_TraccTCP:= TRUE;
	END_IF;
	
(*Robot 25 TraccTCP Request from IC01*)
	IF In_From_ICxx.R25_TraccTCP_Req
		THEN
			Human_Reqs_TraccTCP_R25:= TRUE;		(*Reset at TraccTCP Complete*)
	END_IF;
(*Robot 25 TraccTCP Request*)
	IF MAIN.R25.TraccTCP_Reqd
		THEN
			Robot25_Reqs_TraccTCP:= TRUE;
	END_IF;
	
(*Robot 26 TraccTCP Request from IC01*)
	IF In_From_ICxx.R26_TraccTCP_Req
		THEN
			Human_Reqs_TraccTCP_R26:= TRUE;		(*Reset at TraccTCP Complete*)
	END_IF;
(*Robot 26 TraccTCP Request*)
	IF MAIN.R26.TraccTCP_Reqd
		THEN
			Robot26_Reqs_TraccTCP:= TRUE;
	END_IF;
	
(*Robot 27 TraccTCP Request from IC01*)
	IF In_From_ICxx.R27_TraccTCP_Req
		THEN
			Human_Reqs_TraccTCP_R27:= TRUE;		(*Reset at TraccTCP Complete*)
	END_IF;
(*Robot 27 TraccTCP Request*)
	IF MAIN.R27.TraccTCP_Reqd
		THEN
			Robot27_Reqs_TraccTCP:= TRUE;
	END_IF;
	
(*Robot 28 TraccTCP Request from IC01*)
	IF In_From_ICxx.R28_TraccTCP_Req
		THEN
			Human_Reqs_TraccTCP_R28:= TRUE;		(*Reset at TraccTCP Complete*)
	END_IF;
(*Robot 28 TraccTCP Request*)
	IF MAIN.R28.TraccTCP_Reqd
		THEN
			Robot28_Reqs_TraccTCP:= TRUE;
	END_IF;
	
(*Robot 29 TraccTCP Request from IC01*)
	IF In_From_ICxx.R29_TraccTCP_Req
		THEN
			Human_Reqs_TraccTCP_R29:= TRUE;		(*Reset at TraccTCP Complete*)
	END_IF;
(*Robot 29 TraccTCP Request*)
	IF MAIN.R29.TraccTCP_Reqd
		THEN
			Robot29_Reqs_TraccTCP:= TRUE;
	END_IF;
	
(*Robot 30 TraccTCP Request from IC01*)
	IF In_From_ICxx.R30_TraccTCP_Req
		THEN
			Human_Reqs_TraccTCP_R30:= TRUE;		(*Reset at TraccTCP Complete*)
	END_IF;
(*Robot 30 TraccTCP Request*)
	IF MAIN.R30.TraccTCP_Reqd
		THEN
			Robot30_Reqs_TraccTCP:= TRUE;
	END_IF;
	
(*Gather REQS*)	
	IF Robot1_Reqs_TraccTCP
		OR Robot2_Reqs_TraccTCP
		OR Robot3_Reqs_TraccTCP
		OR Robot4_Reqs_TraccTCP
		OR Robot5_Reqs_TraccTCP
		OR Robot6_Reqs_TraccTCP
		OR Robot7_Reqs_TraccTCP
		OR Robot8_Reqs_TraccTCP
		OR Robot9_Reqs_TraccTCP
		OR Robot10_Reqs_TraccTCP
		OR Robot11_Reqs_TraccTCP
		OR Robot12_Reqs_TraccTCP
		OR Robot13_Reqs_TraccTCP
		OR Robot14_Reqs_TraccTCP
		OR Robot15_Reqs_TraccTCP
		OR Robot16_Reqs_TraccTCP
		OR Robot17_Reqs_TraccTCP
		OR Robot18_Reqs_TraccTCP
		OR Robot19_Reqs_TraccTCP
		OR Robot20_Reqs_TraccTCP
		OR Robot21_Reqs_TraccTCP
		OR Robot22_Reqs_TraccTCP
		OR Robot23_Reqs_TraccTCP
		OR Robot24_Reqs_TraccTCP
		OR Robot25_Reqs_TraccTCP
		OR Robot26_Reqs_TraccTCP
		OR Robot27_Reqs_TraccTCP
		OR Robot28_Reqs_TraccTCP
		OR Robot29_Reqs_TraccTCP
		OR Robot30_Reqs_TraccTCP
		OR In_From_ICxx.Rxx_TraccTCP_Req (*TraccTCP All from UI*)
	THEN
		Robot_Reqs_TraccTCP:= TRUE;
	END_IF;	





(*+++++++++++THIS AREA IS CUSTOM PER INSTALLATION AND WILL HAVE TO BE MODIFIED PER +++++++++++++*)
(*+++++++++++THIS AREA IS CUSTOM PER INSTALLATION AND WILL HAVE TO BE MODIFIED PER +++++++++++++*)

(*$$$$$$$$$$$$$$$$$$$$$$$$$$$$$$$$$$$$$$$$$$$$$$$$ Internal Code $$$$$$$$$$$$$$$$$$$$$$$$$$$$$$$$$$$$$$$$$$$$$$$$$$$$$$$$$$$$$$$$$$$$*)

(*>>>>>>>>>>>>>>>>>>>>>>>>>>>>>>>>>>>>>>>>>> Auto Run Cycle >>>>>>>>>>>>>>>>>>>>>>>>>>>>>>>>>>>>>>>*)
(*+++++++++++THIS AREA IS CUSTOM PER INSTALLATION AND WILL HAVE TO BE MODIFIED PER +++++++++++++*)
(*+++++++++++THIS AREA IS CUSTOM PER INSTALLATION AND WILL HAVE TO BE MODIFIED PER +++++++++++++*)
	(*Control of Auto_Run*)
	Auto_Run:= Enable_Motion AND NOT Cycle_Complete;

	(*Auto Run Enables All Other Auto Cycle Code*)
	IF Auto_Run
		THEN
			(*----------Start Master Test Robots----------*)
			IF NOT Cycle_Complete AND (A_Robot_Reqs_MasterTest OR Human_Reqs_MasterTest)
				THEN
					(*Start All Robots*)
					Start_All_MTRobots:= TRUE;
					(*Allow Robots To Proceed*)
					All_MTRobots_Proceed:= All_Robots_WorkingOK;
			ELSE
					Start_All_MTRobots:= FALSE;
					All_MTRobots_Proceed:= FALSE;
			END_IF;
			(*-------Start Brake Test Robots----------*)
			IF NOT Cycle_Complete AND (All_RobotsReq_BrakeTest OR Human_Reqs_BrakeTest)
					AND NOT Start_All_MTRobots
				THEN
					(*Start All Robots*)
					Start_All_BTRobots:= TRUE;
					(*Allow Robots To Proceed*)
					All_BTRobots_Proceed:= All_Robots_WorkingOK;
			ELSE
					Start_All_BTRobots:= FALSE;
					All_BTRobots_Proceed:= FALSE;
			END_IF;
			(*---------Start Tip Change Robots-------------*)
			IF NOT Cycle_Complete AND (Human_Reqs_TipChange OR Robot_Reqs_TipChange)
					AND NOT Start_All_MTRobots AND NOT Start_All_BTRobots
				THEN
					(*Start All Robots*)
					Start_All_TCRobots:= TRUE;
					(*Allow Robots To Proceed*)
					All_TCRobots_Proceed:= All_Robots_WorkingOK;
			ELSE
					Start_All_TCRobots:= FALSE;
					All_TCRobots_Proceed:= FALSE;
			END_IF;

			(*---------Common Tip Dress-------------*)
			IF NOT Cycle_Complete AND Robot_Reqs_TipDress
					AND NOT Start_All_MTRobots AND NOT Start_All_BTRobots AND NOT Start_All_TCRobots
				THEN
					(*Start All Robots*)
					Start_All_TDRobots:= TRUE;
					(*Allow Robots To Proceed*)
					All_TDRobots_Proceed:= All_Robots_WorkingOK;
			ELSE
					Start_All_TDRobots:= FALSE;
					All_TDRobots_Proceed:= FALSE;
			END_IF;
			
			(*---------Common TraccTCP-------------*) 
			IF NOT Cycle_Complete AND Robot_Reqs_TraccTCP
					AND NOT Start_All_MTRobots AND NOT Start_All_BTRobots AND NOT Start_All_TCRobots
					AND NOT Start_All_TDRobots
				THEN
					(*Start All Robots*)
					Start_All_TraccTCP:= TRUE;
					(*Allow Robots To Proceed*)
					All_TraccTCP_Proceed:= All_Robots_WorkingOK;
			ELSE
					Start_All_TraccTCP:= FALSE;
					All_TraccTCP_Proceed:= FALSE;
			END_IF;

			(*------------Seperated Dresses--------------*)
			(*Robot 1*)
			IF (Robot1_Reqs_TipDress OR Human_Reqs_TipDressR1)
					AND ((NOT Start_All_MTRobots AND NOT Start_All_BTRobots
					AND NOT Start_All_TCRobots AND NOT Start_All_TDRobots)
					OR (MAIN.R1.Task_ID_Ack=Tip_Dress))
				THEN
					(*Start Robot*)
					Start_TDRobot_1:= TRUE;
					(*Allow Robot To Proceed*)
					TDRobot_1_Proceed:= TRUE;
			ELSE
					Start_TDRobot_1:= FALSE;
					TDRobot_1_Proceed:= FALSE;
			END_IF;

			(*Robot 2*)
			IF (Robot2_Reqs_TipDress OR Human_Reqs_TipDressR2)
					AND ((NOT Start_All_MTRobots AND NOT Start_All_BTRobots
					AND NOT Start_All_TCRobots AND NOT Start_All_TDRobots)
					OR (MAIN.R2.Task_ID_Ack=Tip_Dress))
				THEN
					(*Start Robot*)
					Start_TDRobot_2:= TRUE;
					(*Allow Robot To Proceed*)
					TDRobot_2_Proceed:= TRUE;
			ELSE
					Start_TDRobot_2:= FALSE;
					TDRobot_2_Proceed:= FALSE;
			END_IF;

			(*Robot 3*)
			IF (Robot3_Reqs_TipDress OR Human_Reqs_TipDressR3)
					AND ((NOT Start_All_MTRobots AND NOT Start_All_BTRobots
					AND NOT Start_All_TCRobots AND NOT Start_All_TDRobots)
					OR (MAIN.R3.Task_ID_Ack=Tip_Dress))
				THEN
					(*Start Robot*)
					Start_TDRobot_3:= TRUE;
					(*Allow Robot To Proceed*)
					TDRobot_3_Proceed:= TRUE;
			ELSE
					Start_TDRobot_3:= FALSE;
					TDRobot_3_Proceed:= FALSE;
			END_IF;

			(*Robot 4*)
			IF (Robot4_Reqs_TipDress OR Human_Reqs_TipDressR4)
					AND ((NOT Start_All_MTRobots AND NOT Start_All_BTRobots
					AND NOT Start_All_TCRobots AND NOT Start_All_TDRobots)
					OR (MAIN.R4.Task_ID_Ack=Tip_Dress))
				THEN
					(*Start Robot*)
					Start_TDRobot_4:= TRUE;
					(*Allow Robot To Proceed*)
					TDRobot_4_Proceed:= TRUE;
			ELSE
					Start_TDRobot_4:= FALSE;
					TDRobot_4_Proceed:= FALSE;
			END_IF;

			(*Robot 5*)
			IF (Robot5_Reqs_TipDress OR Human_Reqs_TipDressR5)
					AND ((NOT Start_All_MTRobots AND NOT Start_All_BTRobots
					AND NOT Start_All_TCRobots AND NOT Start_All_TDRobots)
					OR (MAIN.R5.Task_ID_Ack=Tip_Dress))
				THEN
					(*Start Robot*)
					Start_TDRobot_5:= TRUE;
					(*Allow Robot To Proceed*)
					TDRobot_5_Proceed:= TRUE;
			ELSE
					Start_TDRobot_5:= FALSE;
					TDRobot_5_Proceed:= FALSE;
			END_IF;

			(*Robot 6*)
			IF (Robot6_Reqs_TipDress OR Human_Reqs_TipDressR6)
					AND ((NOT Start_All_MTRobots AND NOT Start_All_BTRobots
					AND NOT Start_All_TCRobots AND NOT Start_All_TDRobots)
					OR (MAIN.R6.Task_ID_Ack=Tip_Dress))
				THEN
					(*Start Robot*)
					Start_TDRobot_6:= TRUE;
					(*Allow Robot To Proceed*)
					TDRobot_6_Proceed:= TRUE;
			ELSE
					Start_TDRobot_6:= FALSE;
					TDRobot_6_Proceed:= FALSE;
			END_IF;

			(*Robot 7*)
			IF (Robot7_Reqs_TipDress OR Human_Reqs_TipDressR7)
					AND ((NOT Start_All_MTRobots AND NOT Start_All_BTRobots
					AND NOT Start_All_TCRobots AND NOT Start_All_TDRobots)
					OR (MAIN.R7.Task_ID_Ack=Tip_Dress))
				THEN
					(*Start Robot*)
					Start_TDRobot_7:= TRUE;
					(*Allow Robot To Proceed*)
					TDRobot_7_Proceed:= TRUE;
			ELSE
					Start_TDRobot_7:= FALSE;
					TDRobot_7_Proceed:= FALSE;
			END_IF;

			(*Robot 8*)
			IF (Robot8_Reqs_TipDress OR Human_Reqs_TipDressR8)
					AND ((NOT Start_All_MTRobots AND NOT Start_All_BTRobots
					AND NOT Start_All_TCRobots AND NOT Start_All_TDRobots)
					OR (MAIN.R8.Task_ID_Ack=Tip_Dress))
				THEN
					(*Start Robot*)
					Start_TDRobot_8:= TRUE;
					(*Allow Robot To Proceed*)
					TDRobot_8_Proceed:= TRUE;
			ELSE
					Start_TDRobot_8:= FALSE;
					TDRobot_8_Proceed:= FALSE;
			END_IF;

			(*Robot 9*)
			IF (Robot9_Reqs_TipDress OR Human_Reqs_TipDressR9)
					AND ((NOT Start_All_MTRobots AND NOT Start_All_BTRobots
					AND NOT Start_All_TCRobots AND NOT Start_All_TDRobots)
					OR (MAIN.R9.Task_ID_Ack=Tip_Dress))
				THEN
					(*Start Robot*)
					Start_TDRobot_9:= TRUE;
					(*Allow Robot To Proceed*)
					TDRobot_9_Proceed:= TRUE;
			ELSE
					Start_TDRobot_9:= FALSE;
					TDRobot_9_Proceed:= FALSE;
			END_IF;

			(*Robot 10*)
			IF (Robot10_Reqs_TipDress OR Human_Reqs_TipDressR10)
					AND ((NOT Start_All_MTRobots AND NOT Start_All_BTRobots
					AND NOT Start_All_TCRobots AND NOT Start_All_TDRobots)
					OR (MAIN.R10.Task_ID_Ack=Tip_Dress))
				THEN
					(*Start Robot*)
					Start_TDRobot_10:= TRUE;
					(*Allow Robot To Proceed*)
					TDRobot_10_Proceed:= TRUE;
			ELSE
					Start_TDRobot_10:= FALSE;
					TDRobot_10_Proceed:= FALSE;
			END_IF;

			(*Robot 11*)
			IF (Robot11_Reqs_TipDress OR Human_Reqs_TipDressR11)
					AND ((NOT Start_All_MTRobots AND NOT Start_All_BTRobots
					AND NOT Start_All_TCRobots AND NOT Start_All_TDRobots)
					OR (MAIN.R11.Task_ID_Ack=Tip_Dress))
				THEN
					(*Start Robot*)
					Start_TDRobot_11:= TRUE;
					(*Allow Robot To Proceed*)
					TDRobot_11_Proceed:= TRUE;
			ELSE
					Start_TDRobot_11:= FALSE;
					TDRobot_11_Proceed:= FALSE;
			END_IF;

			(*Robot 12*)
			IF (Robot12_Reqs_TipDress OR Human_Reqs_TipDressR12)
					AND ((NOT Start_All_MTRobots AND NOT Start_All_BTRobots
					AND NOT Start_All_TCRobots AND NOT Start_All_TDRobots)
					OR (MAIN.R12.Task_ID_Ack=Tip_Dress))
				THEN
					(*Start Robot*)
					Start_TDRobot_12:= TRUE;
					(*Allow Robot To Proceed*)
					TDRobot_12_Proceed:= TRUE;
			ELSE
					Start_TDRobot_12:= FALSE;
					TDRobot_12_Proceed:= FALSE;
			END_IF;

			(*Robot 13*)
			IF (Robot13_Reqs_TipDress OR Human_Reqs_TipDressR13)
					AND ((NOT Start_All_MTRobots AND NOT Start_All_BTRobots
					AND NOT Start_All_TCRobots AND NOT Start_All_TDRobots)
					OR (MAIN.R13.Task_ID_Ack=Tip_Dress))
				THEN
					(*Start Robot*)
					Start_TDRobot_13:= TRUE;
					(*Allow Robot To Proceed*)
					TDRobot_13_Proceed:= TRUE;
			ELSE
					Start_TDRobot_13:= FALSE;
					TDRobot_13_Proceed:= FALSE;
			END_IF;

			(*Robot 14*)
			IF (Robot14_Reqs_TipDress OR Human_Reqs_TipDressR14)
					AND ((NOT Start_All_MTRobots AND NOT Start_All_BTRobots
					AND NOT Start_All_TCRobots AND NOT Start_All_TDRobots)
					OR (MAIN.R14.Task_ID_Ack=Tip_Dress))
				THEN
					(*Start Robot*)
					Start_TDRobot_14:= TRUE;
					(*Allow Robot To Proceed*)
					TDRobot_14_Proceed:= TRUE;
			ELSE
					Start_TDRobot_14:= FALSE;
					TDRobot_14_Proceed:= FALSE;
			END_IF;

			(*Robot 15*)
			IF (Robot15_Reqs_TipDress OR Human_Reqs_TipDressR15)
					AND ((NOT Start_All_MTRobots AND NOT Start_All_BTRobots
					AND NOT Start_All_TCRobots AND NOT Start_All_TDRobots)
					OR (MAIN.R15.Task_ID_Ack=Tip_Dress))
				THEN
					(*Start Robot*)
					Start_TDRobot_15:= TRUE;
					(*Allow Robot To Proceed*)
					TDRobot_15_Proceed:= TRUE;
			ELSE
					Start_TDRobot_15:= FALSE;
					TDRobot_15_Proceed:= FALSE;
			END_IF;

			(*Robot 16*)
			IF (Robot16_Reqs_TipDress OR Human_Reqs_TipDressR16)
					AND ((NOT Start_All_MTRobots AND NOT Start_All_BTRobots
					AND NOT Start_All_TCRobots AND NOT Start_All_TDRobots)
					OR (MAIN.R16.Task_ID_Ack=Tip_Dress))
				THEN
					(*Start Robot*)
					Start_TDRobot_16:= TRUE;
					(*Allow Robot To Proceed*)
					TDRobot_16_Proceed:= TRUE;
			ELSE
					Start_TDRobot_16:= FALSE;
					TDRobot_16_Proceed:= FALSE;
			END_IF;

			(*Robot 17*)
			IF (Robot17_Reqs_TipDress OR Human_Reqs_TipDressR17)
					AND ((NOT Start_All_MTRobots AND NOT Start_All_BTRobots
					AND NOT Start_All_TCRobots AND NOT Start_All_TDRobots)
					OR (MAIN.R17.Task_ID_Ack=Tip_Dress))
				THEN
					(*Start Robot*)
					Start_TDRobot_17:= TRUE;
					(*Allow Robot To Proceed*)
					TDRobot_17_Proceed:= TRUE;
			ELSE
					Start_TDRobot_17:= FALSE;
					TDRobot_17_Proceed:= FALSE;
			END_IF;

			(*Robot 18*)
			IF (Robot18_Reqs_TipDress OR Human_Reqs_TipDressR18)
					AND ((NOT Start_All_MTRobots AND NOT Start_All_BTRobots
					AND NOT Start_All_TCRobots AND NOT Start_All_TDRobots)
					OR (MAIN.R18.Task_ID_Ack=Tip_Dress))
				THEN
					(*Start Robot*)
					Start_TDRobot_18:= TRUE;
					(*Allow Robot To Proceed*)
					TDRobot_18_Proceed:= TRUE;
			ELSE
					Start_TDRobot_18:= FALSE;
					TDRobot_18_Proceed:= FALSE;
			END_IF;

			(*Robot 19*)
			IF (Robot19_Reqs_TipDress OR Human_Reqs_TipDressR19)
					AND ((NOT Start_All_MTRobots AND NOT Start_All_BTRobots
					AND NOT Start_All_TCRobots AND NOT Start_All_TDRobots)
					OR (MAIN.R19.Task_ID_Ack=Tip_Dress))
				THEN
					(*Start Robot*)
					Start_TDRobot_19:= TRUE;
					(*Allow Robot To Proceed*)
					TDRobot_19_Proceed:= TRUE;
			ELSE
					Start_TDRobot_19:= FALSE;
					TDRobot_19_Proceed:= FALSE;
			END_IF;

			(*Robot 20*)
			IF (Robot20_Reqs_TipDress OR Human_Reqs_TipDressR20)
					AND ((NOT Start_All_MTRobots AND NOT Start_All_BTRobots
					AND NOT Start_All_TCRobots AND NOT Start_All_TDRobots)
					OR (MAIN.R20.Task_ID_Ack=Tip_Dress))
				THEN
					(*Start Robot*)
					Start_TDRobot_20:= TRUE;
					(*Allow Robot To Proceed*)
					TDRobot_20_Proceed:= TRUE;
			ELSE
					Start_TDRobot_20:= FALSE;
					TDRobot_20_Proceed:= FALSE;
			END_IF;

			(*Robot 21*)
			IF (Robot21_Reqs_TipDress OR Human_Reqs_TipDressR21)
					AND ((NOT Start_All_MTRobots AND NOT Start_All_BTRobots
					AND NOT Start_All_TCRobots AND NOT Start_All_TDRobots)
					OR (MAIN.R21.Task_ID_Ack=Tip_Dress))
				THEN
					(*Start Robot*)
					Start_TDRobot_21:= TRUE;
					(*Allow Robot To Proceed*)
					TDRobot_20_Proceed:= TRUE;
			ELSE
					Start_TDRobot_21:= FALSE;
					TDRobot_21_Proceed:= FALSE;
			END_IF;

			(*Robot 22*)
			IF (Robot22_Reqs_TipDress OR Human_Reqs_TipDressR22)
					AND ((NOT Start_All_MTRobots AND NOT Start_All_BTRobots
					AND NOT Start_All_TCRobots AND NOT Start_All_TDRobots)
					OR (MAIN.R22.Task_ID_Ack=Tip_Dress))
				THEN
					(*Start Robot*)
					Start_TDRobot_22:= TRUE;
					(*Allow Robot To Proceed*)
					TDRobot_22_Proceed:= TRUE;
			ELSE
					Start_TDRobot_22:= FALSE;
					TDRobot_22_Proceed:= FALSE;
			END_IF;

			(*Robot 23*)
			IF (Robot23_Reqs_TipDress OR Human_Reqs_TipDressR23)
					AND ((NOT Start_All_MTRobots AND NOT Start_All_BTRobots
					AND NOT Start_All_TCRobots AND NOT Start_All_TDRobots)
					OR (MAIN.R23.Task_ID_Ack=Tip_Dress))
				THEN
					(*Start Robot*)
					Start_TDRobot_23:= TRUE;
					(*Allow Robot To Proceed*)
					TDRobot_23_Proceed:= TRUE;
			ELSE
					Start_TDRobot_23:= FALSE;
					TDRobot_23_Proceed:= FALSE;
			END_IF;

			(*Robot 24*)
			IF (Robot24_Reqs_TipDress OR Human_Reqs_TipDressR24)
					AND ((NOT Start_All_MTRobots AND NOT Start_All_BTRobots
					AND NOT Start_All_TCRobots AND NOT Start_All_TDRobots)
					OR (MAIN.R24.Task_ID_Ack=Tip_Dress))
				THEN
					(*Start Robot*)
					Start_TDRobot_24:= TRUE;
					(*Allow Robot To Proceed*)
					TDRobot_24_Proceed:= TRUE;
			ELSE
					Start_TDRobot_24:= FALSE;
					TDRobot_24_Proceed:= FALSE;
			END_IF;

			(*Robot 25*)
			IF (Robot25_Reqs_TipDress OR Human_Reqs_TipDressR25)
					AND ((NOT Start_All_MTRobots AND NOT Start_All_BTRobots
					AND NOT Start_All_TCRobots AND NOT Start_All_TDRobots)
					OR (MAIN.R25.Task_ID_Ack=Tip_Dress))
				THEN
					(*Start Robot*)
					Start_TDRobot_25:= TRUE;
					(*Allow Robot To Proceed*)
					TDRobot_25_Proceed:= TRUE;
			ELSE
					Start_TDRobot_25:= FALSE;
					TDRobot_25_Proceed:= FALSE;
			END_IF;

			(*Robot 26*)
			IF (Robot26_Reqs_TipDress OR Human_Reqs_TipDressR26)
					AND ((NOT Start_All_MTRobots AND NOT Start_All_BTRobots
					AND NOT Start_All_TCRobots AND NOT Start_All_TDRobots)
					OR (MAIN.R26.Task_ID_Ack=Tip_Dress))
				THEN
					(*Start Robot*)
					Start_TDRobot_26:= TRUE;
					(*Allow Robot To Proceed*)
					TDRobot_26_Proceed:= TRUE;
			ELSE
					Start_TDRobot_26:= FALSE;
					TDRobot_26_Proceed:= FALSE;
			END_IF;

			(*Robot 27*)
			IF (Robot27_Reqs_TipDress OR Human_Reqs_TipDressR27)
					AND ((NOT Start_All_MTRobots AND NOT Start_All_BTRobots
					AND NOT Start_All_TCRobots AND NOT Start_All_TDRobots)
					OR (MAIN.R27.Task_ID_Ack=Tip_Dress))
				THEN
					(*Start Robot*)
					Start_TDRobot_27:= TRUE;
					(*Allow Robot To Proceed*)
					TDRobot_27_Proceed:= TRUE;
			ELSE
					Start_TDRobot_27:= FALSE;
					TDRobot_27_Proceed:= FALSE;
			END_IF;

			(*Robot 28*)
			IF (Robot28_Reqs_TipDress OR Human_Reqs_TipDressR28)
					AND ((NOT Start_All_MTRobots AND NOT Start_All_BTRobots
					AND NOT Start_All_TCRobots AND NOT Start_All_TDRobots)
					OR (MAIN.R28.Task_ID_Ack=Tip_Dress))
				THEN
					(*Start Robot*)
					Start_TDRobot_28:= TRUE;
					(*Allow Robot To Proceed*)
					TDRobot_28_Proceed:= TRUE;
			ELSE
					Start_TDRobot_28:= FALSE;
					TDRobot_28_Proceed:= FALSE;
			END_IF;

			(*Robot 29*)
			IF (Robot29_Reqs_TipDress OR Human_Reqs_TipDressR29)
					AND ((NOT Start_All_MTRobots AND NOT Start_All_BTRobots
					AND NOT Start_All_TCRobots AND NOT Start_All_TDRobots)
					OR (MAIN.R29.Task_ID_Ack=Tip_Dress))
				THEN
					(*Start Robot*)
					Start_TDRobot_29:= TRUE;
					(*Allow Robot To Proceed*)
					TDRobot_29_Proceed:= TRUE;
			ELSE
					Start_TDRobot_29:= FALSE;
					TDRobot_29_Proceed:= FALSE;
			END_IF;

			(*Robot 30*)
			IF (Robot30_Reqs_TipDress OR Human_Reqs_TipDressR30)
					AND ((NOT Start_All_MTRobots AND NOT Start_All_BTRobots
					AND NOT Start_All_TCRobots AND NOT Start_All_TDRobots)
					OR (MAIN.R30.Task_ID_Ack=Tip_Dress))
				THEN
					(*Start Robot*)
					Start_TDRobot_30:= TRUE;
					(*Allow Robot To Proceed*)
					TDRobot_30_Proceed:= TRUE;
			ELSE
					Start_TDRobot_30:= FALSE;
					TDRobot_30_Proceed:= FALSE;
			END_IF;

			(*------------------Separated TraccTCP------------------*)			
			(*Robot 1*)
			IF (Human_Reqs_TraccTCP_R1)
					AND ((NOT Start_All_MTRobots AND NOT Start_All_BTRobots
					AND NOT Start_All_TCRobots AND NOT Start_All_TDRobots)
					OR (MAIN.R1.Task_ID_Ack=Tracc_TCP))
				THEN
					(*Start Robot*)
					Start_TraccTCP_1:= TRUE;
					(*Allow Robot to Proceed*)
					TraccRobot_1_Proceed:= TRUE;
			ELSE
					Start_TraccTCP_1:= FALSE;
					TraccRobot_1_Proceed:= FALSE;
			END_IF;
				
			(*Robot 2*)
			IF (Human_Reqs_TraccTCP_R2)
					AND ((NOT Start_All_MTRobots AND NOT Start_All_BTRobots
					AND NOT Start_All_TCRobots AND NOT Start_All_TDRobots)
					OR (MAIN.R2.Task_ID_Ack=Tracc_TCP))
				THEN
					(*Start Robot*)
					Start_TraccTCP_2:= TRUE;
					(*Allow Robot to Proceed*)
					TraccRobot_2_Proceed:= TRUE;
			ELSE
					Start_TraccTCP_2:= FALSE;
					TraccRobot_2_Proceed:= FALSE;		
			END_IF;
			
			(*Robot 3*)
			IF (Human_Reqs_TraccTCP_R3)
					AND ((NOT Start_All_MTRobots AND NOT Start_All_BTRobots
					AND NOT Start_All_TCRobots AND NOT Start_All_TDRobots)
					OR (MAIN.R3.Task_ID_Ack=Tracc_TCP))
				THEN
					(*Start Robot*)
					Start_TraccTCP_3:= TRUE;
					(*Allow Robot to Proceed*)
					TraccRobot_3_Proceed:= TRUE;
			ELSE
					Start_TraccTCP_3:= FALSE;
					TraccRobot_3_Proceed:= FALSE;
			END_IF;
			
			(*Robot 4*)
			IF (Human_Reqs_TraccTCP_R4)
					AND ((NOT Start_All_MTRobots AND NOT Start_All_BTRobots
					AND NOT Start_All_TCRobots AND NOT Start_All_TDRobots)
					OR (MAIN.R4.Task_ID_Ack=Tracc_TCP))
				THEN
					(*Start Robot*)
					Start_TraccTCP_4:= TRUE;
					(*Allow Robot to Proceed*)
					TraccRobot_4_Proceed:= TRUE;
			ELSE
					Start_TraccTCP_4:= FALSE;
					TraccRobot_4_Proceed:= FALSE;
			END_IF;	
			
			(*Robot 5*)
			IF (Human_Reqs_TraccTCP_R5)
					AND ((NOT Start_All_MTRobots AND NOT Start_All_BTRobots
					AND NOT Start_All_TCRobots AND NOT Start_All_TDRobots)
					OR (MAIN.R5.Task_ID_Ack=Tracc_TCP))
				THEN
					(*Start Robot*)
					Start_TraccTCP_5:= TRUE;
					(*Allow Robot to Proceed*)
					TraccRobot_5_Proceed:= TRUE;
			ELSE
					Start_TraccTCP_5:= FALSE;
					TraccRobot_5_Proceed:= FALSE;
			END_IF;	
			
			(*Robot 6*)
			IF (Human_Reqs_TraccTCP_R6)
					AND ((NOT Start_All_MTRobots AND NOT Start_All_BTRobots
					AND NOT Start_All_TCRobots AND NOT Start_All_TDRobots)
					OR (MAIN.R6.Task_ID_Ack=Tracc_TCP))
				THEN
					(*Start Robot*)
					Start_TraccTCP_6:= TRUE;
					(*Allow Robot to Proceed*)
					TraccRobot_6_Proceed:= TRUE;
			ELSE
					Start_TraccTCP_6:= FALSE;
					TraccRobot_6_Proceed:= FALSE;
			END_IF;	
			
			(*Robot 7*)
			IF (Human_Reqs_TraccTCP_R7)
					AND ((NOT Start_All_MTRobots AND NOT Start_All_BTRobots
					AND NOT Start_All_TCRobots AND NOT Start_All_TDRobots)
					OR (MAIN.R7.Task_ID_Ack=Tracc_TCP))
				THEN
					(*Start Robot*)
					Start_TraccTCP_7:= TRUE;
					(*Allow Robot to Proceed*)
					TraccRobot_7_Proceed:= TRUE;
			ELSE
					Start_TraccTCP_7:= FALSE;
					TraccRobot_7_Proceed:= FALSE;
			END_IF;	
			
			(*Robot 8*)
			IF (Human_Reqs_TraccTCP_R8)
					AND ((NOT Start_All_MTRobots AND NOT Start_All_BTRobots
					AND NOT Start_All_TCRobots AND NOT Start_All_TDRobots)
					OR (MAIN.R8.Task_ID_Ack=Tracc_TCP))
				THEN
					(*Start Robot*)
					Start_TraccTCP_8:= TRUE;
					(*Allow Robot to Proceed*)
					TraccRobot_8_Proceed:= TRUE;
			ELSE
					Start_TraccTCP_8:= FALSE;
					TraccRobot_8_Proceed:= FALSE;
			END_IF;	
			
			(*Robot 9*)
			IF (Human_Reqs_TraccTCP_R9)
					AND ((NOT Start_All_MTRobots AND NOT Start_All_BTRobots
					AND NOT Start_All_TCRobots AND NOT Start_All_TDRobots)
					OR (MAIN.R9.Task_ID_Ack=Tracc_TCP))
				THEN
					(*Start Robot*)
					Start_TraccTCP_9:= TRUE;
					(*Allow Robot to Proceed*)
					TraccRobot_9_Proceed:= TRUE;
			ELSE
					Start_TraccTCP_9:= FALSE;
					TraccRobot_9_Proceed:= FALSE;
			END_IF;	
			
			(*Robot 10*)
			IF (Human_Reqs_TraccTCP_R10)
					AND ((NOT Start_All_MTRobots AND NOT Start_All_BTRobots
					AND NOT Start_All_TCRobots AND NOT Start_All_TDRobots)
					OR (MAIN.R10.Task_ID_Ack=Tracc_TCP))
				THEN
					(*Start Robot*)
					Start_TraccTCP_10:= TRUE;
					(*Allow Robot to Proceed*)
					TraccRobot_10_Proceed:= TRUE;
			ELSE
					Start_TraccTCP_10:= FALSE;
					TraccRobot_10_Proceed:= FALSE;
			END_IF;	
			
			(*Robot 11*)
			IF (Human_Reqs_TraccTCP_R11)
					AND ((NOT Start_All_MTRobots AND NOT Start_All_BTRobots
					AND NOT Start_All_TCRobots AND NOT Start_All_TDRobots)
					OR (MAIN.R11.Task_ID_Ack=Tracc_TCP))
				THEN
					(*Start Robot*)
					Start_TraccTCP_11:= TRUE;
					(*Allow Robot to Proceed*)
					TraccRobot_11_Proceed:= TRUE;
			ELSE
					Start_TraccTCP_11:= FALSE;
					TraccRobot_11_Proceed:= FALSE;
			END_IF;	
			
			(*Robot 12*)
			IF (Human_Reqs_TraccTCP_R12)
					AND ((NOT Start_All_MTRobots AND NOT Start_All_BTRobots
					AND NOT Start_All_TCRobots AND NOT Start_All_TDRobots)
					OR (MAIN.R12.Task_ID_Ack=Tracc_TCP))
				THEN
					(*Start Robot*)
					Start_TraccTCP_12:= TRUE;
					(*Allow Robot to Proceed*)
					TraccRobot_12_Proceed:= TRUE;
			ELSE
					Start_TraccTCP_12:= FALSE;
					TraccRobot_12_Proceed:= FALSE;
			END_IF;	
			
			(*Robot 13*)
			IF (Human_Reqs_TraccTCP_R13)
					AND ((NOT Start_All_MTRobots AND NOT Start_All_BTRobots
					AND NOT Start_All_TCRobots AND NOT Start_All_TDRobots)
					OR (MAIN.R13.Task_ID_Ack=Tracc_TCP))
				THEN
					(*Start Robot*)
					Start_TraccTCP_13:= TRUE;
					(*Allow Robot to Proceed*)
					TraccRobot_13_Proceed:= TRUE;
			ELSE
					Start_TraccTCP_13:= FALSE;
					TraccRobot_13_Proceed:= FALSE;
			END_IF;	
			
			(*Robot 14*)
			IF (Human_Reqs_TraccTCP_R14)
					AND ((NOT Start_All_MTRobots AND NOT Start_All_BTRobots
					AND NOT Start_All_TCRobots AND NOT Start_All_TDRobots)
					OR (MAIN.R14.Task_ID_Ack=Tracc_TCP))
				THEN
					(*Start Robot*)
					Start_TraccTCP_14:= TRUE;
					(*Allow Robot to Proceed*)
					TraccRobot_14_Proceed:= TRUE;
			ELSE
					Start_TraccTCP_14:= FALSE;
					TraccRobot_14_Proceed:= FALSE;
			END_IF;	
			
			(*Robot 15*)
			IF (Human_Reqs_TraccTCP_R15)
					AND ((NOT Start_All_MTRobots AND NOT Start_All_BTRobots
					AND NOT Start_All_TCRobots AND NOT Start_All_TDRobots)
					OR (MAIN.R15.Task_ID_Ack=Tracc_TCP))
				THEN
					(*Start Robot*)
					Start_TraccTCP_15:= TRUE;
					(*Allow Robot to Proceed*)
					TraccRobot_15_Proceed:= TRUE;
			ELSE
					Start_TraccTCP_15:= FALSE;
					TraccRobot_15_Proceed:= FALSE;
			END_IF;	
			
			(*Robot 16*)
			IF (Human_Reqs_TraccTCP_R16)
					AND ((NOT Start_All_MTRobots AND NOT Start_All_BTRobots
					AND NOT Start_All_TCRobots AND NOT Start_All_TDRobots)
					OR (MAIN.R16.Task_ID_Ack=Tracc_TCP))
				THEN
					(*Start Robot*)
					Start_TraccTCP_16:= TRUE;
					(*Allow Robot to Proceed*)
					TraccRobot_16_Proceed:= TRUE;
			ELSE
					Start_TraccTCP_16:= FALSE;
					TraccRobot_16_Proceed:= FALSE;
			END_IF;	
			
			(*Robot 17*)
			IF (Human_Reqs_TraccTCP_R4)
					AND ((NOT Start_All_MTRobots AND NOT Start_All_BTRobots
					AND NOT Start_All_TCRobots AND NOT Start_All_TDRobots)
					OR (MAIN.R17.Task_ID_Ack=Tracc_TCP))
				THEN
					(*Start Robot*)
					Start_TraccTCP_17:= TRUE;
					(*Allow Robot to Proceed*)
					TraccRobot_17_Proceed:= TRUE;
			ELSE
					Start_TraccTCP_17:= FALSE;
					TraccRobot_17_Proceed:= FALSE;
			END_IF;	
			
			(*Robot 18*)
			IF (Human_Reqs_TraccTCP_R18)
					AND ((NOT Start_All_MTRobots AND NOT Start_All_BTRobots
					AND NOT Start_All_TCRobots AND NOT Start_All_TDRobots)
					OR (MAIN.R18.Task_ID_Ack=Tracc_TCP))
				THEN
					(*Start Robot*)
					Start_TraccTCP_18:= TRUE;
					(*Allow Robot to Proceed*)
					TraccRobot_18_Proceed:= TRUE;
			ELSE
					Start_TraccTCP_18:= FALSE;
					TraccRobot_18_Proceed:= FALSE;
			END_IF;	
			
			(*Robot 19*)
			IF (Human_Reqs_TraccTCP_R19)
					AND ((NOT Start_All_MTRobots AND NOT Start_All_BTRobots
					AND NOT Start_All_TCRobots AND NOT Start_All_TDRobots)
					OR (MAIN.R19.Task_ID_Ack=Tracc_TCP))
				THEN
					(*Start Robot*)
					Start_TraccTCP_19:= TRUE;
					(*Allow Robot to Proceed*)
					TraccRobot_19_Proceed:= TRUE;
			ELSE
					Start_TraccTCP_19:= FALSE;
					TraccRobot_19_Proceed:= FALSE;
			END_IF;	
			
			(*Robot 20*)
			IF (Human_Reqs_TraccTCP_R20)
					AND ((NOT Start_All_MTRobots AND NOT Start_All_BTRobots
					AND NOT Start_All_TCRobots AND NOT Start_All_TDRobots)
					OR (MAIN.R20.Task_ID_Ack=Tracc_TCP))
				THEN
					(*Start Robot*)
					Start_TraccTCP_20:= TRUE;
					(*Allow Robot to Proceed*)
					TraccRobot_20_Proceed:= TRUE;
			ELSE
					Start_TraccTCP_20:= FALSE;
					TraccRobot_20_Proceed:= FALSE;
			END_IF;	
			
